{attribute 'object_name' := 'CycleStartDuty'}
METHOD PROTECTED CycleStartDuty : BOOL
// ----------------------------------------------------------------------------------
// cyclic actions outside of statemachine

// Simulation active
IF (SIf.stCfg.bolSimulation) THEN
	;
ELSE
	;
END_IF

// Cyclic call of the client connection
fbClientConnection();
// Cyclic call of method "HandleRxData"
THIS^.HandleRxData();

// Generate socket connected status info
IF (fbClientConnection.eState = eSOCKET_CONNECTED) THEN
	SIf.stStatus.bolSocketConnected:= TRUE;
ELSE
	SIf.stStatus.bolSocketConnected:= FALSE;	
	SIf.stStatus.bolComChecked:= FALSE;
END_IF

// Command close socket can be executed all the time.
// Used for error recovery in case if parent controller has an error.
IF (SIf.intCmd=cBCD_CMD_CLOSE_SOCKET) THEN	
	stStateMachine.intStateNext := cBCD_STA_CloseSocketBusy;
END_IF
			
SIf.strCmd := THIS^.getCmdState(intCmdState:=SIf.intCmd,bolState:=FALSE);
END_METHOD

{attribute 'object_name' := 'FB_init'}
METHOD FB_init : BOOL
VAR_INPUT
	///if TRUE, the retain variables are initialized (warm start / cold start)
	bInitRetains: BOOL;
	///if TRUE, the instance afterwards gets moved into the copy code (online change)
	bInCopyCode: BOOL;
END_VAR
// Communication Settings
SIf.stCfg.strSensorIPAdr := '192.168.1.103';  //'192.168.0.10'; 
SIf.stCfg.udiSensorPort := 9004;
SIf.stCfg.bolResponseIncludingDiagnostics := FALSE;
SIf.stCfg.iSensorType := E_BCD_Type.KEYENCE;

// Parameter
SIf.stPar.tTOConnection := T#50S;
SIf.stPar.tTOReceive := T#5S;
SIf.stPar.tTOSend := T#5S;
END_METHOD

{attribute 'object_name' := 'getCmdState'}
METHOD PROTECTED getCmdState : STRING
VAR_INPUT
	intCmdState: INT;
	bolState: BOOL;
END_VAR
// get string cmd/state string information in runtime
IF (bolState=FALSE) THEN
	
// cmd's
	CASE intCmdState OF
		cBCD_CMD_DONE: 
			getCmdState := 'cBCD_CMD_DONE';
		cBCD_CMD_CONNECT_SOCKET: 
			getCmdState := 'cBCD_CMD_CONNECT_SOCKET';
		cBCD_CMD_CLOSE_SOCKET: 
			getCmdState := 'cBCD_CMD_CLOSE_SOCKET';
		cBCD_CMD_READ_BARCODE: 
			getCmdState := 'cBCD_CMD_READ_BARCODE';		
		cBCD_CMD_COM_TEST: 
			getCmdState := 'cBCD_CMD_COM_TEST';			
	END_CASE;
ELSE

// state's
	CASE intCmdState OF
		cBCD_STA_WaitForJob: 
			getCmdState := 'cBCD_STA_WaitForJob';
		cBCD_STA_ConnectSocketBusy: 
			getCmdState := 'cBCD_STA_ConnectSocketBusy';
		cBCD_STA_CloseSocketBusy: 
			getCmdState := 'cBCD_STA_CloseSocketBusy';
		cBCD_STA_SocketClosed: 
			getCmdState := 'cBCD_STA_SocketClosed';	
		cBCD_STA_ReadCodeBusy: 
			getCmdState := 'cBCD_STA_ReadCodeBusy';	
		cBCD_STA_ComTestBusy:
			getCmdState := 'cBCD_STA_ComTestBusy';	
		cBCD_STA_Error: 
			getCmdState := 'cBCD_STA_Error';
	END_CASE;
	
END_IF
END_METHOD

{attribute 'object_name' := 'getSIf'}
METHOD getSIf : POINTER TO T_BCD
getSIf := ADR(SIf);
END_METHOD

{attribute 'object_name' := 'HandleRxData'}
METHOD PRIVATE HandleRxData
VAR
	uinI: UINT;
END_VAR
// GET/FETCH RX DATA
CASE intRxState OF
	
	// wait for read command
	cRxIdle:
		IF (bolExecuteRead=TRUE) AND (fbClientConnection.eState = eSOCKET_CONNECTED)THEN	

			// clear rx buffer
			FOR uinI:= 0 TO SIZEOF(aRxData)-1 DO
				aRxData[uinI]:= 16#00;
			END_FOR
			// Delete last message
			strReceivedMessage:= '';
			udiReceivedBytes := 0;
								
			// receive frame			
			fbReceive( bExecute := FALSE );
			fbReceive( 	sSrvNetId	:= '',
						hSocket		:= fbClientConnection.hSocket,
						cbLen		:= SIZEOF(aRxData),
						pDest		:= ADR(aRxData),
						bExecute	:= TRUE,
						tTimeout	:= SIf.stPar.tTOReceive);
			intRxState := cRxBusy;		
		END_IF
		
	// wait until receive not busy
	cRxBusy:
		fbReceive( bExecute := FALSE );
		IF NOT fbReceive.bBusy THEN
			IF NOT fbReceive.bError THEN
				IF (fbReceive.nRecBytes > 0) THEN (* some bytes received *)
					udiReceivedBytes := fbReceive.nRecBytes;
					intRxState := cRxConv; // convert received message
				ELSE
					// Try to read again
					intRxState := cRxIdle;
				END_IF	
			// Error	
			ELSE
				IF (SIf.stErr.bolErrorActive = FALSE) THEN
					SIf.stErr.bolErrorActive := TRUE;	
					SIf.stErr.udiErrorID := fbReceive.nErrId;	
					// Try to close the socket. Needs reconnect for socket after an error!	
					stStateMachine.intStateNext := cBCD_STA_CloseSocketBusy;	
				END_IF	
			END_IF			
		END_IF
			
	// convert received message to string
	cRxConv: 
		THIS^.PrepareReadMsg();
		THIS^.CheckSensorError(); // Error response: [STX]sFA <x>[ETX]    	
		bolExecuteRead:= FALSE; // Read done and data converted to string format
		intRxState := cRxIdle;
		
END_CASE
END_METHOD

{attribute 'object_name' := 'HandleTxData'}
METHOD PRIVATE HandleTxData
// HANDLE TX DATA
CASE intTxState OF
	
	// wait for send command (ready for send)
	cTxIdle:
		IF (bolExecuteSend) AND (fbClientConnection.eState = eSOCKET_CONNECTED)THEN									
			// send frame
			fbSend( bExecute := FALSE );
			fbSend(	sSrvNetID 	:= '',
					hSocket		:= fbClientConnection.hSocket,
					cbLen		:= rTxData.intMessageSize,
					pSrc		:= ADR(rTxData.aTxData),					// pointer to the frame data
					bExecute	:= TRUE,
					tTimeout 	:= SIf.stPar.tTOSend);
	
			intTxState := cTxBusy;							
		END_IF
		
	// wait until send not busy
	cTxBusy:
		fbSend( bExecute := FALSE );
		IF NOT (fbSend.bBusy) THEN
			intTxState := cTxIdle;
			// Check about FUB error	
			IF (fbSend.bError = TRUE) THEN
				IF (SIf.stErr.bolErrorActive = FALSE) THEN
					SIf.stErr.bolErrorActive := TRUE;	
					SIf.stErr.udiErrorID := fbSend.nErrId;	
					// Try to close the socket. Needs reconnect for socket after an error!	
					stStateMachine.intStateNext := cBCD_STA_CloseSocketBusy;	
				END_IF				
			// no error
			ELSE
				udiNSend := udiNSend + 1; // increment the number of send frames
				bolExecuteSend:= FALSE;
			END_IF
		END_IF
		
END_CASE
END_METHOD

{attribute 'object_name' := 'PrepareBarCodeData'}
METHOD PRIVATE PrepareBarCodeData
VAR
	intI: INT;
	intStartIndex: INT;
	intStartIndexCode: INT;
	bASCIISign: BYTE;
	strCharacter: STRING(1);
END_VAR

// Note: Currently only the bar code is read out from the received message. "OI=" section in message.
// Other data sections like e.g. "TT=", "OTL=", "CC=" are not prepared.

// ----------------------------------------------------
// Get bar code and write result to structure "stData"
// ----------------------------------------------------
	
// Example of message: <stx> <CR><LF> TT=125ms OTL=0mm CC=1 OI=25<CR><LF>45376049874<CR><LF> .... and so on ...   <etx>
				 
// Get start index for bar code 'OI='
intStartIndex := TC2_STANDARD.FIND(strReceivedMessage,'OI=');

// Loop over received message to get the bar code
FOR intI:=intStartIndex TO LEN(strReceivedMessage)-intStartIndex DO	
	// Convert to ASCII to detect CR and LF
	bASCIISign:= F_ToASC(Mid(strReceivedMessage,1,intI));
	// The bar code number starts after LF					
	IF (bASCIISign = cLF) THEN
		// Save start index of the bar code
		intStartIndexCode:= intI + 1;
	END_IF
	// Read every single number of the bar code until the end "CR"
	IF ((intStartIndexCode <> 0) AND (intI >= intStartIndexCode)) THEN
		// As long as the end is not reached...(The bar code number ends with CR)	
		IF (bASCIISign <> cCR) THEN								
			// Write result to structure stData	
			strCharacter:= Mid(strReceivedMessage,1,intI);
			SIf.stData.strBarCode:= CONCAT(SIf.stData.strBarCode,strCharacter);	
			SIf.stData.uliBarCode:= STRING_TO_ULINT(SIf.stData.strBarCode);
			SIf.stData.bolCodeReaded:= TRUE;																	
		ELSE
			// end of bar code reached "CR" -> EXIT loop
			EXIT;
		END_IF
	END_IF
	
END_FOR
END_METHOD

{attribute 'object_name' := 'PrepareReadMsg'}
METHOD PRIVATE PrepareReadMsg
VAR
	uinI: UINT;
	strCharacter: STRING(1);
END_VAR
// Delete last message
strReceivedMessage:= '';

// Loop over receive buffer
FOR uinI:= 0 TO SIZEOF(aRxData)-1 DO	
	// Start of text?
	IF (aRxData[uinI] = cSTX) THEN
		;
	// End of text?
	ELSIF (aRxData[uinI] = cETX) THEN
		EXIT;
	ELSE
		// Convert ASCII to string
		strCharacter:= F_ToCHR(aRxData[uinI]);
		strReceivedMessage:= CONCAT(strReceivedMessage,strCharacter);			
	END_IF
END_FOR
END_METHOD

{attribute 'object_name' := 'PrepareSendMsg'}
METHOD PRIVATE PrepareSendMsg
VAR_INPUT
	strMsg: STRING;
END_VAR
VAR
	intI: UINT;
	strCharacter: STRING(1);
END_VAR
// Clear send buffer
ClearTxBuffer();

// STX - start of telegramm
rTxData.aTxData[0]:= cSTX;

// Loop over message string and convert to ASCII
FOR intI:= 1 TO INT_TO_UINT(LEN(strMsg)) DO
	// Get char
	strCharacter:= MID(strMsg,1,UINT_TO_INT(intI));
	// Convert to ASCII
	rTxData.aTxData[intI]:= F_ToASC(strCharacter);
END_FOR

// ETX - end of telegramm
rTxData.aTxData[intI]:= cETX;

rTxData.intMessageSize := intI + 1;
END_METHOD

{attribute 'object_name' := 'sta_CloseSocketBusy'}
METHOD PROTECTED sta_CloseSocketBusy : BOOL
// state implemetation
//--------------------------------------------------------------------------------------
// Entry action
	IF (stStateMachine.intState<>stStateMachine.intStateLastCycle) THEN
		stStateMachine.intStateHistory := stStateMachine.intStateLastCycle;
		stStateMachine.intStateLastCycle := stStateMachine.intState;
		
		// Reset pending commands			
		bolExecuteSend:= FALSE;
		bolExecuteRead:= FALSE;
		// Reset Rx/Tx states
		intRxState:= cRxIdle;
		intTxState:= cTxIdle;
		// Close socket
		fbClientConnection.bEnable:= FALSE;

	END_IF

//--------------------------------------------------------------------------------------
// Cyclic action
	IF (stStateMachine.intState=stStateMachine.intStateLastCycle) THEN
		
	
		// State Change Condition

		// Check about FUB error	
		IF (fbClientConnection.bError = TRUE) OR (fbClientConnection.nErrId <> 0) THEN
			SIf.stErr.bolErrorActive := TRUE;	
			SIf.stErr.bolSocketError := TRUE;
			SIf.stErr.udiErrorID := fbClientConnection.nErrId;
			stStateMachine.intStateNext := cBCD_STA_Error;
		END_IF
	
		// Wait until socket is closed	
		IF (fbClientConnection.eState = eSOCKET_CLOSED) THEN
			stStateMachine.intStateNext := cBCD_STA_WaitForJob;
		ELSIF  (SIf.stErr.bolErrorActive= TRUE) THEN 
			stStateMachine.intStateNext := cBCD_STA_Error;		
		END_IF
	
	END_IF

//--------------------------------------------------------------------------------------
// Exit action
	IF (stStateMachine.intState<>stStateMachine.intStateNext) THEN
		SIf.intCmd := cBCD_CMD_DONE;
	END_IF
END_METHOD

{attribute 'object_name' := 'sta_ComTestBusy'}
METHOD PROTECTED sta_ComTestBusy : BOOL
// state implemetation
//--------------------------------------------------------------------------------------
// Entry action
	IF (stStateMachine.intState<>stStateMachine.intStateLastCycle) THEN
		stStateMachine.intStateHistory := stStateMachine.intStateLastCycle;
		stStateMachine.intStateLastCycle := stStateMachine.intState;

		// Clear data
		SIf.stData.stDevInfo.strComTestResult:='';
		SIf.stStatus.bolComChecked:=FALSE;
	
		// Init sub state machine
		stSubStateMachine.intState := cBCD_SUB_Send;
		stSubStateMachine.intStateNext := cBCD_SUB_Send;	
	END_IF

//--------------------------------------------------------------------------------------
// Cyclic action
	IF (stStateMachine.intState=stStateMachine.intStateLastCycle) THEN
			
		// sub state machine for reading the bar code	
		CASE stSubStateMachine.intState OF

			cBCD_SUB_Send:
				// Check Tx state idle
				IF (intTxState = cTxIdle) THEN
					CASE SIf.stCfg.iSensorType OF
						E_BCD_Type.SICK:
							THIS^.PrepareSendMsg('sRI0'); // Call SOPAS command "sRI0"
							
						E_BCD_Type.KEYENCE:
							THIS^.PrepareSendMsg('BCLR'); // clear send buffer
					END_CASE
					bolExecuteSend:= TRUE;
					stSubStateMachine.intState := cBCD_SUB_Wait;
				END_IF
		
			cBCD_SUB_Wait:
				// Wait until executed -> flag set back to false by method handle TxData
				IF (bolExecuteSend=FALSE)THEN
					stSubStateMachine.intState := cBCD_SUB_Read;
				END_IF
				
			cBCD_SUB_Read:
				// Check Rx state idle
				IF (intRxState = cRxIdle) THEN
					bolExecuteRead:= TRUE;
					stSubStateMachine.intState := cBCD_SUB_CheckAnswer;
				END_IF
			
			cBCD_SUB_CheckAnswer:
				// Wait until executed -> flag set back to false by method handle RxData
				IF (bolExecuteRead=FALSE)THEN				
					// Check about corresponding answer for the command	
					CASE SIf.stCfg.iSensorType OF
						E_BCD_Type.SICK:					
							IF (TC2_STANDARD.FIND(strReceivedMessage,'sRA') <> 0) THEN
								SIf.stData.stDevInfo.strComTestResult:=strReceivedMessage;
								SIf.stStatus.bolComChecked:=TRUE;
							END_IF
						
						E_BCD_Type.KEYENCE:
							IF (TC2_STANDARD.FIND(strReceivedMessage,'OK,BCLR') <> 0) THEN
								SIf.stData.stDevInfo.strComTestResult:=strReceivedMessage;
								SIf.stStatus.bolComChecked:=TRUE;
							END_IF
					END_CASE
					stSubStateMachine.intState := cBCD_SUB_Done;
				END_IF
			
			cBCD_SUB_Done:
				; // job executed
			
		END_CASE
		
		 // job executed
		IF (stSubStateMachine.intState = cBCD_SUB_Done) THEN
			stStateMachine.intStateNext := cBCD_STA_WaitForJob;	
		END_IF
	
	END_IF

//--------------------------------------------------------------------------------------
// Exit action
	IF (stStateMachine.intState<>stStateMachine.intStateNext) THEN
		SIf.intCmd := cBCD_CMD_DONE;
	END_IF
END_METHOD

{attribute 'object_name' := 'sta_ConnectSocketBusy'}
METHOD PROTECTED sta_ConnectSocketBusy : BOOL
// state implemetation
//--------------------------------------------------------------------------------------
// Entry action
	IF (stStateMachine.intState<>stStateMachine.intStateLastCycle) THEN
		stStateMachine.intStateHistory := stStateMachine.intStateLastCycle;
		stStateMachine.intStateLastCycle := stStateMachine.intState;
			
		// Initialize and connect socket
		fbClientConnection.nMode := CONNECT_MODE_ENABLEDBG; 			// not used
		fbClientConnection.sRemoteHost := SIf.stCfg.strSensorIPAdr;
		fbClientConnection.nRemotePort := SIf.stCfg.udiSensorPort;
		fbClientConnection.tReconnect := SIf.stPar.tTOConnection;
		fbClientConnection.bEnable:= TRUE;

	END_IF

//--------------------------------------------------------------------------------------
// Cyclic action
	IF (stStateMachine.intState=stStateMachine.intStateLastCycle) THEN
		
	
		// State Change Condition

		// Check about FUB error	
		IF (fbClientConnection.bError = TRUE) OR (fbClientConnection.nErrId <> 0) THEN
			SIf.stErr.bolErrorActive := TRUE;	
			SIf.stErr.bolSocketError := TRUE;
			SIf.stErr.udiErrorID := fbClientConnection.nErrId;
			stStateMachine.intStateNext := cBCD_STA_Error;
		END_IF
	
		// Wait for socket handle ID	
		IF (fbClientConnection.hSocket.handle <> 0) AND (fbClientConnection.eState = eSOCKET_CONNECTED) THEN
			stStateMachine.intStateNext := cBCD_STA_WaitForJob;
		END_IF

	END_IF

//--------------------------------------------------------------------------------------
// Exit action
	IF (stStateMachine.intState<>stStateMachine.intStateNext) THEN
		SIf.intCmd := cBCD_CMD_DONE;
	END_IF
END_METHOD

{attribute 'object_name' := 'sta_Error'}
METHOD PROTECTED sta_Error : BOOL
// state implemetation
//--------------------------------------------------------------------------------------
// Entry action
	IF (stStateMachine.intState<>stStateMachine.intStateLastCycle) THEN
		stStateMachine.intStateHistory := stStateMachine.intStateLastCycle;
		stStateMachine.intStateLastCycle := stStateMachine.intState;
		
		// Reset pending commands			
		bolExecuteSend:= FALSE;
		bolExecuteRead:= FALSE;
		// Reset Rx/Tx states
		intRxState:= cRxIdle;
		intTxState:= cTxIdle;
		
	END_IF


//--------------------------------------------------------------------------------------
// Cyclic action
	IF (stStateMachine.intState=stStateMachine.intStateLastCycle) THEN
			
		// State Change Condition
		IF (SIf.stErr.bolErrAck = TRUE) THEN
			// Reset all active errors
			SIf.stErr.bolErrorActive := FALSE;
			SIf.stErr.bolSocketError := FALSE;
			SIf.stErr.bolSensorError := FALSE;
			SIf.stErr.udiErrorID := 0;
			SIf.stErr.bolErrAck := FALSE;
			// Needs reconnect for socket after an error!		
			stStateMachine.intStateNext := cBCD_STA_CloseSocketBusy;		
		END_IF
		
	END_IF

//--------------------------------------------------------------------------------------
// Exit action
	IF (stStateMachine.intState<>stStateMachine.intStateNext) THEN
		;
	END_IF
END_METHOD

{attribute 'object_name' := 'sta_ReadCodeBusy'}
METHOD PROTECTED sta_ReadCodeBusy : BOOL
// state implemetation
//--------------------------------------------------------------------------------------
// Entry action
	IF (stStateMachine.intState<>stStateMachine.intStateLastCycle) THEN
		stStateMachine.intStateHistory := stStateMachine.intStateLastCycle;
		stStateMachine.intStateLastCycle := stStateMachine.intState;
		
		// Clear data
		SIf.stData.uliBarCode:=0;
		SIf.stData.strBarCode:='';
		SIf.stData.bolCodeReaded:= FALSE;
						
		// Init sub state machine
		stSubStateMachine.intState := cBCD_SUB_Send;
		stSubStateMachine.intStateNext := cBCD_SUB_Send;	
	END_IF

//--------------------------------------------------------------------------------------
// Cyclic action
	IF (stStateMachine.intState=stStateMachine.intStateLastCycle) THEN
			
		// sub state machine for reading the bar code	
		CASE stSubStateMachine.intState OF

			cBCD_SUB_Send:
				// Check Tx state idle
				IF (intTxState = cTxIdle) THEN
					CASE SIf.stCfg.iSensorType OF
						E_BCD_Type.SICK:
							THIS^.PrepareSendMsg('sMN mTCgateon'); // Call SOPAS method "sMN mTCgateon"
							bolExecuteSend:= TRUE;
							stSubStateMachine.intState := cBCD_SUB_Wait;
							
						E_BCD_Type.KEYENCE:
							THIS^.PrepareSendMsg('LON'); // Call Trigger ON
							bolExecuteSend:= TRUE;
							stSubStateMachine.intState := cBCD_SUB_Wait;
					ELSE
						SIf.stData.strBarCode:= 'no sensor type defined';
						SIf.stData.uliBarCode:= 0;
					END_CASE
					
				END_IF
		
			cBCD_SUB_Wait:
				// Wait until executed -> flag set back to false by method handle TxData
				IF (bolExecuteSend=FALSE)THEN
					stSubStateMachine.intState := cBCD_SUB_Read;
				END_IF
				
			cBCD_SUB_Read:
				// Check Rx state idle
				IF (intRxState = cRxIdle) THEN
					bolExecuteRead:= TRUE;
					stSubStateMachine.intState := cBCD_SUB_CheckAnswer;
				END_IF
			
			cBCD_SUB_CheckAnswer:
				// Wait until executed -> flag set back to false by method handle RxData
				IF (bolExecuteRead=FALSE)THEN				
					// Check about corresponding answer for the called method
					CASE SIf.stCfg.iSensorType OF
						E_BCD_Type.SICK:
							IF (FC_StrComp(strReceivedMessage,'sAN mTCgateon 1') = 0) THEN			
								// Check Rx state idle
								IF (intRxState = cRxIdle) THEN
									bolExecuteRead:= TRUE;
									stSubStateMachine.intState := cBCD_SUB_GetData;
								END_IF
							END_IF
							
						E_BCD_Type.KEYENCE:
							IF (FC_StrComp(strReceivedMessage,'OK,LON') = 0) THEN			
								// Check Rx state idle
								IF (intRxState = cRxIdle) THEN
									bolExecuteRead:= TRUE;
									stSubStateMachine.intState := cBCD_SUB_GetData;
								END_IF
							END_IF
					END_CASE
				END_IF
			
			cBCD_SUB_GetData:
				// Wait until executed -> flag set back to false by method handle RxData
				IF (bolExecuteRead=FALSE)THEN
					
					CASE SIf.stCfg.iSensorType OF
						E_BCD_Type.SICK:
							// No barcode recognized after the end of the time window ("duration" setting of sensor object trigger), NoRead !
							IF (((TC2_STANDARD.FIND(strReceivedMessage,'OI=') <> 0) OR NOT SIf.stCfg.bolResponseIncludingDiagnostics) 
								AND (TC2_STANDARD.FIND(strReceivedMessage,'*NoRead*') <> 0)) THEN			
								SIf.stData.strBarCode:='NoRead';
								stSubStateMachine.intState := cBCD_SUB_Done;
							END_IF
							
							// Barcode detected within the time window
							IF (((TC2_STANDARD.FIND(strReceivedMessage,'OI=') <> 0) OR NOT SIf.stCfg.bolResponseIncludingDiagnostics) 
								AND NOT (TC2_STANDARD.FIND(strReceivedMessage,'*NoRead*') <> 0)) THEN			
								// Prepare bar code data from received message
								THIS^.PrepareBarCodeData();
								stSubStateMachine.intState := cBCD_SUB_Done;
							END_IF
						
						E_BCD_Type.KEYENCE:
							// No barcode recognized after the end of the time window ("duration" setting of sensor object trigger), NoRead !
							IF (TC2_STANDARD.FIND(strReceivedMessage,'ERROR') <> 0) THEN			
								SIf.stData.strBarCode:='NoRead';
								stSubStateMachine.intState := cBCD_SUB_Done;
							END_IF
							
							// Barcode detected within the time window
							IF NOT (TC2_STANDARD.FIND(strReceivedMessage,'ERROR') <> 0) THEN			
								// Prepare bar code data from received message
								iStringLength := Tc2_Standard.LEN(strReceivedMessage);
								SIf.stData.strBarCode := Tc2_Standard.LEFT(strReceivedMessage,iStringLength-1);
								SIf.stData.uliBarCode:= STRING_TO_ULINT(SIf.stData.strBarCode);
								stSubStateMachine.intState := cBCD_SUB_Done;
							END_IF
					END_CASE
				END_IF
			
			cBCD_SUB_Done:
				; // job executed
			
		END_CASE
		
		 // job executed
		IF (stSubStateMachine.intState = cBCD_SUB_Done) THEN
			stStateMachine.intStateNext := cBCD_STA_WaitForJob;	
		END_IF
			
	END_IF

//--------------------------------------------------------------------------------------
// Exit action
	IF (stStateMachine.intState<>stStateMachine.intStateNext) THEN
		SIf.intCmd := cBCD_CMD_DONE;
	END_IF
END_METHOD

{attribute 'object_name' := 'sta_SocketClosed'}
METHOD PROTECTED sta_SocketClosed : BOOL
// state implemetation
//--------------------------------------------------------------------------------------
// Entry action
	IF (stStateMachine.intState<>stStateMachine.intStateLastCycle) THEN
		stStateMachine.intStateLastCycle := stStateMachine.intState;
		;
	END_IF

//--------------------------------------------------------------------------------------
// Cyclic action
	IF (stStateMachine.intState=stStateMachine.intStateLastCycle) THEN

		// State Change Condition
		IF (SIf.intCmd=cBCD_CMD_CONNECT_SOCKET) THEN
			stStateMachine.intStateNext := cBCD_STA_ConnectSocketBusy;
		END_IF
		
	END_IF

//--------------------------------------------------------------------------------------
// Exit action
	IF (stStateMachine.intState<>stStateMachine.intStateNext) THEN
		;
	END_IF
END_METHOD

{attribute 'object_name' := 'sta_WaitForJob'}
METHOD PROTECTED sta_WaitForJob : BOOL
// state implemetation
//--------------------------------------------------------------------------------------
// Entry action
	IF (stStateMachine.intState<>stStateMachine.intStateLastCycle) THEN
		stStateMachine.intStateLastCycle := stStateMachine.intState;
	END_IF


//--------------------------------------------------------------------------------------
// Cyclic action
	IF (stStateMachine.intState=stStateMachine.intStateLastCycle) THEN

		// State Change Condition
		IF (SIf.intCmd=cBCD_CMD_CONNECT_SOCKET) THEN						// Connect TCP socket
			stStateMachine.intStateNext := cBCD_STA_ConnectSocketBusy;
		ELSIF (SIf.intCmd=cBCD_CMD_CLOSE_SOCKET) THEN						// Close TCP socket
			stStateMachine.intStateNext := cBCD_STA_CloseSocketBusy;
		ELSIF (SIf.intCmd=cBCD_CMD_COM_TEST) THEN							// Communication test 
			stStateMachine.intStateNext := cBCD_STA_ComTestBusy;	
		ELSIF (SIf.intCmd=cBCD_CMD_READ_BARCODE) THEN						// Read bar code
			stStateMachine.intStateNext := cBCD_STA_ReadCodeBusy;				
		END_IF

				
	END_IF

//--------------------------------------------------------------------------------------
// Exit action
	IF (stStateMachine.intState<>stStateMachine.intStateNext) THEN
		;
	END_IF
END_METHOD

{attribute 'object_name' := 'StateMachine'}
METHOD PROTECTED StateMachine : BOOL

// main statemachine
CASE stStateMachine.intState OF	
	cBCD_STA_WaitForJob:
   		THIS^.sta_WaitForJob();
	cBCD_STA_ConnectSocketBusy: 
        THIS^.sta_ConnectSocketBusy();	
	cBCD_STA_CloseSocketBusy: 
        THIS^.sta_CloseSocketBusy();		
	cBCD_STA_SocketClosed: 
        THIS^.sta_SocketClosed();	
	cBCD_STA_ComTestBusy:
	    THIS^.sta_ComTestBusy();
	cBCD_STA_ReadCodeBusy:
	    THIS^.sta_ReadCodeBusy();
    cBCD_STA_Error: 
        THIS^.sta_Error();
END_CASE;
END_METHOD

END_FUNCTION_BLOCK

// POUs/Controller/Driver/BCD (Bar code driver)/FC_StrComp
FUNCTION FC_StrComp : DINT
VAR_INPUT
	strArg1: STRING(255);
	strArg2: STRING(255);
END_VAR
VAR
	stArg1: TC2_UTILITIES.T_Arg;
	stArg2: TC2_UTILITIES.T_Arg;
END_VAR


// String compare function use F_ARGCMP from beckhoff lib. TC2_UTILITIES

// set parameter for arg1
stArg1.cbLen:= INT_TO_UDINT(TC2_STANDARD.LEN(strArg1));
stArg1.pData:= ADR(strArg1);
stArg1.eType:= ARGTYPE_STRING;

// set parameter for arg2
stArg2.cbLen:= INT_TO_UDINT(TC2_STANDARD.LEN(strArg2));
stArg2.pData:= ADR(strArg2);
stArg2.eType:= ARGTYPE_STRING;

// call F_ARGCMP
FC_StrComp:= TC2_UTILITIES.F_ARGCMP(TRUE,stArg1,stArg2);

END_FUNCTION

// POUs/Controller/Driver/PRS [Present Sensor]/FB_PRS
FUNCTION_BLOCK FB_PRS EXTENDS FB_CtrlBase
VAR_INPUT
	In_bolPresent				: BOOL;
END_VAR
VAR_OUTPUT
	Out_bolPresent				: BOOL;
END_VAR
VAR
	/// Specific interface struct for public access
	SIf					: T_Ctrl_SIf_PRS;
END_VAR

(*__________________________________________________________________________________________________
¦	
¦	Vistaprint Schweiz GmbH
¦	CH - 8401 Winterthur
¦
¦	www.vistaprint.ch - info@vistaprint.ch
¦___________________________________________________________________________________________________

Function desription:
Vacuum Pump implementation. 


History:
Version		Date			Author		Comment
---------------------------------------------------------------------------------------------------
0.00.1		09.07.2013		PC			Start history
___________________________________________________________________________________________________*)


IF (me.bolActivate) THEN // cyclic call enabled
	IF (CIf.Info.bolInitDone=FALSE) THEN // first cycle -> init
		CtrlInit();
		CIf.Info.bolInitDone := TRUE;
	ELSE
		CycleStartDuty();
	
		Always();
		
		StateMachine();
		
		CycleEndDuty();
	END_IF
END_IF;

METHOD PROTECTED Always : BOOL
SUPER^.Always();

// ----------------------------------------------------------------------------------
// cyclic actions outside of statemachine
IF (me.StateMachine.intState<>cSTA_SINGLE_ANSWER) THEN
	
	; // always error supervision
	
END_IF

// ----------------------------------------------------------------------------------
// Conditions Always
IF (((me.Alarm.eActivAlmClass=E_AlmClass.EOFF) OR (me.Alarm.eActivAlmClass=E_AlmClass.OFF) OR (me.intCmd=cCMD_OFF))
		 AND (me.StateMachine.intState<>cSTA_ERROR) AND (me.StateMachine.intState<>cSTA_ERRORQuit) AND
		(me.StateMachine.intState<>cSTA_OFF) AND (me.StateMachine.intState<>cSTA_OFFBusy)) THEN
	// alarm evt EOFF, OFF or cmd off
	me.StateMachine.intStateNext := cSTA_OFFBusy;
END_IF
END_METHOD

PROPERTY PUBLIC CtrlSIf : POINTER TO T_CTRL_SIf_PRS
GET
CtrlSIf := ADR(SIf);
END_GET
END_PROPERTY

METHOD FB_init : BOOL
VAR_INPUT
	bInitRetains : BOOL; // if TRUE, the retain variables are initialized (warm start / cold start)
	bInCopyCode : BOOL;  // if TRUE, the instance afterwards gets moved into the copy code (online change)
END_VAR
VAR
	iIdx		: UINT;
	iLength		: UINT;	
END_VAR
//------------------------------------------------------------------------------------------------------------------------
// to manually change in new FUB implementation!!!
// define valid commands for this controller
iLength := SIZEOF(CIf.Job.aCmdList)/SIZEOF(CIf.Job.aCmdList[0]);
iIdx := 0;

WHILE (iIdx < iLength) AND (CIf.Job.aCmdList[iIdx].intCmd <> cCMD_INITIALIZED) DO
	iIdx := iIdx + 1; 
END_WHILE

IF (iIdx < iLength) THEN
// Add configuration of own comands	
	;
ELSE
	// Error if the aCmdList Array is to small
END_IF

// set name of class/typ
CIf.Info.strType := 'FB_PRS';
CIf.Info.strFullName := 'Present Sensor';

// set alarm class

//*******************************************************************************
// initial values
//*******************************************************************************

// software configuration
CIf.SwCfg.bolExist := TRUE;
CIf.SwCfg.bolEnable := TRUE;
CIf.SwCfg.bolSimulation :=  FALSE;

// parameter
SIf.Par.bolSimHangerAvailable := FALSE;
SIf.Par.udiDebounceAbsentTime_ms := 100;
SIf.Par.udiDebouncePresentTime_ms := 1500;
END_METHOD

METHOD PROTECTED getCmdState : STRING

VAR_INPUT
	intCmdState: INT;
	bolState: BOOL;
END_VAR
getCmdState := SUPER^.getCmdState(intCmdState:=intCmdState,bolState:=bolState); // get global/base defined cmds/states

IF (getCmdState='') THEN // global not defined get local
	// get string cmd/state string information in runtime
	IF (bolState=FALSE) THEN
		;
	ELSE
		// States's
		CASE intCmdState OF
			PRS_CmdState.cSTA_ABSENT: 
				getCmdState := 'cSTA_ABSENT';
			PRS_CmdState.cSTA_ABSENTBusy: 
				getCmdState := 'cSTA_ABSENTBusy';
			PRS_CmdState.cSTA_PRESENT: 
				getCmdState := 'cSTA_PRESENT';
			PRS_CmdState.cSTA_PRESENTBusy: 
				getCmdState := 'cSTA_PRESENTBusy';
		END_CASE;
	END_IF
END_IF
END_METHOD

METHOD getCtrlSIf : POINTER TO T_Ctrl_SIf_PRS
getCtrlSIf := ADR(SIf);
END_METHOD

METHOD PROTECTED IoInBridge : BOOL
// digitale and analoge inputs read from hardware or forcing
SIf.In.bolPresent.map := THIS^.In_bolPresent;

IF (CIf.SwCfg.bolSimulation = FALSE) THEN
	getInBol(CIf.Job.bolIoForce,ADR(SIf.In.bolPresent));
ELSE
	//simulation of global IO
END_IF
END_METHOD

METHOD PROTECTED IoOutBridge : BOOL
VAR
	bolSwitchValvesOff: BOOL;
END_VAR
// digitale and analoge inputs read from hardware or forcing
IF (CIf.SwCfg.bolSimulation = FALSE) THEN
//	setOutBol(CIf.Job.bolIoForce ,ADR(SIf.Out.bolClose));
	;
//	THIS^.Out_bolClose := SIf.Out.bolClose.map;
END_IF
END_METHOD

METHOD PROTECTED sta_ABSENT : BOOL
VAR_INPUT
END_VAR
// state implemetation
//--------------------------------------------------------------------------------------
// Entry action
	IF (me.StateMachine.intState<>me.StateMachine.intStateLastCycle) THEN
		me.StateMachine.intStateLastCycle := me.StateMachine.intState;
		THIS^.Out_bolPresent := FALSE;
	END_IF


//--------------------------------------------------------------------------------------
// Cyclic action
	IF (me.StateMachine.intState=me.StateMachine.intStateLastCycle) THEN
		IF CIf.SwCfg.bolSimulation THEN
			IF SIf.Par.bolSimHangerAvailable THEN
				me.StateMachine.intStateNext := PRS_CmdState.cSTA_PRESENTBusy;
			END_IF
		ELSE
			IF SIf.In.bolPresent.intern  THEN
				me.StateMachine.intStateNext := PRS_CmdState.cSTA_PRESENTBusy;
			END_IF;		
		END_IF
	END_IF


//--------------------------------------------------------------------------------------
// Exit action
	IF (me.StateMachine.intState<>me.StateMachine.intStateNext) THEN
		;
	END_IF
END_METHOD

METHOD PROTECTED sta_ABSENTBusy : BOOL
VAR_INPUT
END_VAR
// state implemetation
//--------------------------------------------------------------------------------------
// Entry action
	IF (me.StateMachine.intState<>me.StateMachine.intStateLastCycle) THEN
		me.StateMachine.intStateLastCycle := me.StateMachine.intState;
	END_IF


//--------------------------------------------------------------------------------------
// Cyclic action
	IF (me.StateMachine.intState=me.StateMachine.intStateLastCycle) THEN
		IF CIf.SwCfg.bolSimulation THEN
			IF SIf.Par.bolSimHangerAvailable THEN
				me.StateMachine.intStateNext := PRS_CmdState.cSTA_PRESENT;
			END_IF
		ELSE
			IF SIf.In.bolPresent.intern  THEN
				me.StateMachine.intStateNext := PRS_CmdState.cSTA_PRESENT;
			END_IF;		
			
			IF NOT SIf.In.bolPresent.intern AND (me.StateMachine.udiTimeInState_ms > SIf.Par.udiDebounceAbsentTime_ms) THEN
				me.StateMachine.intStateNext :=  PRS_CmdState.cSTA_ABSENT;
			END_IF
		END_IF
	END_IF


//--------------------------------------------------------------------------------------
// Exit action
	IF (me.StateMachine.intState<>me.StateMachine.intStateNext) THEN
		;
	END_IF
END_METHOD

METHOD PROTECTED sta_PON : BOOL
VAR_INPUT
END_VAR
// state implemetation
//--------------------------------------------------------------------------------------
// Entry action
	IF (me.StateMachine.intState<>me.StateMachine.intStateLastCycle) THEN
		me.StateMachine.intStateLastCycle := me.StateMachine.intState;
		
	END_IF


//--------------------------------------------------------------------------------------
// Cyclic action
	IF (me.StateMachine.intState=me.StateMachine.intStateLastCycle) THEN
		me.StateMachine.intStateNext := PRS_CmdState.cSTA_ABSENTBusy;
	END_IF




//--------------------------------------------------------------------------------------
// Exit action
	IF (me.StateMachine.intState<>me.StateMachine.intStateNext) THEN
		;
	END_IF
END_METHOD

METHOD PROTECTED sta_PRESENT : BOOL
VAR_INPUT
END_VAR
// state implemetation
//--------------------------------------------------------------------------------------
// Entry action
	IF (me.StateMachine.intState<>me.StateMachine.intStateLastCycle) THEN
		me.StateMachine.intStateLastCycle := me.StateMachine.intState;
		THIS^.Out_bolPresent := TRUE;
	END_IF


//--------------------------------------------------------------------------------------
// Cyclic action
	IF (me.StateMachine.intState=me.StateMachine.intStateLastCycle) THEN
		IF CIf.SwCfg.bolSimulation THEN
			IF NOT SIf.Par.bolSimHangerAvailable THEN
				me.StateMachine.intStateNext := PRS_CmdState.cSTA_ABSENTBusy;
			END_IF
		ELSE
			IF NOT SIf.In.bolPresent.intern  THEN
				me.StateMachine.intStateNext := PRS_CmdState.cSTA_ABSENTBusy;
			END_IF;		
		END_IF
	END_IF


//--------------------------------------------------------------------------------------
// Exit action
	IF (me.StateMachine.intState<>me.StateMachine.intStateNext) THEN
		;
	END_IF
END_METHOD

METHOD PROTECTED sta_PRESENTBusy : BOOL
VAR_INPUT
END_VAR
// state implemetation
//--------------------------------------------------------------------------------------
// Entry action
	IF (me.StateMachine.intState<>me.StateMachine.intStateLastCycle) THEN
		me.StateMachine.intStateLastCycle := me.StateMachine.intState;
	END_IF


//--------------------------------------------------------------------------------------
// Cyclic action
	IF (me.StateMachine.intState=me.StateMachine.intStateLastCycle) THEN
		IF CIf.SwCfg.bolSimulation THEN
			IF NOT SIf.Par.bolSimHangerAvailable THEN
				me.StateMachine.intStateNext := PRS_CmdState.cSTA_ABSENT;
			END_IF
		ELSE
			IF NOT SIf.In.bolPresent.intern  THEN
				me.StateMachine.intStateNext := PRS_CmdState.cSTA_ABSENT;
			END_IF;		
			
			IF SIf.In.bolPresent.intern AND (me.StateMachine.udiTimeInState_ms > SIf.Par.udiDebouncePresentTime_ms) THEN
				me.StateMachine.intStateNext :=  PRS_CmdState.cSTA_PRESENT;
			END_IF
		END_IF
	END_IF


//--------------------------------------------------------------------------------------
// Exit action
	IF (me.StateMachine.intState<>me.StateMachine.intStateNext) THEN
		;
	END_IF
END_METHOD

METHOD PROTECTED StateMachine : BOOL
SUPER^.StateMachine();

// main statemachine of base controller
CASE me.StateMachine.intState OF
    PRS_CmdState.cSTA_ABSENT: 
        THIS^.sta_ABSENT();
    PRS_CmdState.cSTA_ABSENTBusy: 
        THIS^.sta_ABSENTBusy();
    PRS_CmdState.cSTA_PRESENT: 
        THIS^.sta_PRESENT();
    PRS_CmdState.cSTA_PRESENTBusy: 
        THIS^.sta_PRESENTBusy();
END_CASE;
END_METHOD

END_FUNCTION_BLOCK

// POUs/Controller/Driver/RFD (RFID Driver)/FB_Com_3964R
FUNCTION_BLOCK FB_Com_3964R
VAR_INPUT
	/// Pointer to Received Data Array
	In_pRxData: POINTER TO ARRAY[0..255] OF BYTE;
	/// Pointer to Sending Data Array
	In_pTxData: POINTER TO ARRAY[0..255] OF BYTE;
	/// Amounth of sending data
	In_udiTxCount: UDINT;
	/// Error Acknowledge 
	In_bolErrorAck: BOOL;
END_VAR
VAR_IN_OUT
	/// Command to send Data 1=command; 0=Done
	InOut_bolSend: BOOL;
	/// Command Data received 1=received; 0=Done=Ready for next Data
	InOut_bolRec: BOOL;
END_VAR
VAR_OUTPUT
	/// Amounth of received data
	Out_udiRxCount: UDINT;
	/// Serial interface communication error
	Out_bolComError: BOOL;
	/// Error in protocoll procedure
	Out_bolProtocolErr: BOOL;
	/// Error information to master
	Out_udiErrorCode: UDINT;
END_VAR
VAR
	In_stEL6inData AT %I*: TC2_SERIALCOM.EL6inData22B;
	Out_stEL6outData AT %Q*: TC2_SERIALCOM.EL6outData22B;
	/// Internal Variables
	udiI: UDINT;
	/// Local variable for loops
	udiK: UDINT;
	/// Internal Error Reset
	bolIntReset: BOOL;
	/// Count call trials
	uinCountCall: UINT;
	/// Count call Retrys
	uinCountRetry: UINT;
	/// Temporary value for cecking the sum
	bytCheckValue: BYTE;
	/// Antenna is initializied, until it is not initializied, it send 16#02 in all possible baudrates
	bolSLGInitialized: BOOL := FALSE;
	/// Check Timeout
	bolTimeout: BOOL;
	/// Check Timeout
	bolWait: BOOL;
	/// Send NAK needed
	bolSendNAK: BOOL;
	/// Receive Wait signs
	timWaitReceive: TIME := TIME#5ms;
	/// Receive Wait signs
	timWaitAck: TIME := TIME#400ms;
	/// Sign delay time
	timZVZ: TIME := TIME#45ms;
	/// Time ACK delay
	timQVZ: TIME := TIME#145ms;
	/// Initialisation of the HW card
	bolInitRequest: BOOL;
	/// Setting of the HW Card
	bolSendContinious: BOOL;
	/// Priority at RFID
	bolPriority: BOOL;
	/// Send DLE doubletimes
	bolDLEDouble: BOOL;
	/// New data received
	bolComDataReceived: BOOL;
	/// receiving busy
	bolComRecBusy: BOOL;
	/// Received Data
	udiComSizeReceiveData: UDINT;
	/// Sending busy
	bolComSendBusy: BOOL;
	/// Error at serial line control
	bolErrSerialLineControl: BOOL;
	/// Error at serial line control
	stErrSerialLineControl: ComError_t;
	/// Error at serial line  receiving data
	bolErrReceive: BOOL;
	/// Error at serial line  receiving data
	stErrReceive: ComError_t;
	/// Error at serial line sending data
	bolErrSend: BOOL;
	/// Error at serial line sending data
	stErrSend: ComError_t;
	/// Define Buffer for preparations
	aRxData: ARRAY[0..255] OF BYTE;
	aTxData: ARRAY[0..255] OF BYTE;
	/// Define Buffer for Funciton
	stRxBuffer: TC2_SERIALCOM.ComBuffer;
	/// Transmit data buffer; used with all receive function blocks 
	stTxBuffer: TC2_SERIALCOM.ComBuffer;
	/// Sub Statemachine
	intState: INT := 0;
	intStateOld: INT := 0;
	udiStateLoop: UDINT;
	a_intStateHist: ARRAY[0..9] OF INT;
	udiStateDebug: UDINT;
	udiStateDebugMax: UDINT;
	/// Function for serial communication
	fbSerialLineControl: TC2_SERIALCOM.SerialLineControl;
	fbSerialReceiveData: TC2_SERIALCOM.ReceiveData;
	fbSerialSendData: TC2_SERIALCOM.SendData;
	fbSerialClearComBuffer: TC2_SERIALCOM.ClearComBuffer;
	fbTon: TC2_STANDARD.TON;
	fbWait: TC2_STANDARD.TON;
	fbZVZ: TC2_STANDARD.TON;
	fbQVZ: TC2_STANDARD.TON;
	fbPriority: TC2_STANDARD.TON;
END_VAR
VAR CONSTANT
	cSTX: USINT := 16#2;
	cDLE: USINT := 16#10;
	cETX: USINT := 16#3;
	cNAK: USINT := 16#15;
	/// Startup
	cRFD_3964_Start: INT := 2500;
	/// Startup
	cRFD_3964_Init: INT := 2501;
	/// Wait for Job
	cRFD_3964_Wait: INT := 2502;
	/// Read recived sign
	cRFD_3964_RxRead: INT := 2504;
	/// Ackn. receiving ready
	cRFD_3964_RxReadRdy: INT := 2506;
	/// Recive Data
	cRFD_3964_RxData: INT := 2508;
	/// Achn. received Data
	cRFD_3964_RxCheckData: INT := 2510;
	/// Send Ack to Slave
	cRFD_3964_RxAck: INT := 2512;
	/// Send Ack to Slave
	cRFD_3964_RxAck2: INT := 2514;
	/// Send Request to Slave
	cRFD_3964_TxRequest: INT := 2550;
	/// Send Wait answer
	cRFD_3964_TxWait: INT := 2552;
	/// Send Data
	cRFD_3964_TxSend: INT := 2554;
	/// Send Wait for Ack
	cRFD_3964_TxAck: INT := 2556;
	/// Error
	cRFD_3964_Error: INT := 2580;
END_VAR

(*__________________________________________________________________________________________________
¦	
¦	Vistaprint Schweiz GmbH
¦	CH - 8401 Winterthur
¦
¦	www.vistaprint.ch - info@vistaprint.ch
¦___________________________________________________________________________________________________

Function desription:
Driver for communication protocoll 3964R
Description in Siemens manual from CP341, A5E02191070-03


History:
Version		Date			Author		Comment
---------------------------------------------------------------------------------------------------
0.00.1		23.07.2013		AVME/PRE	Start history
___________________________________________________________________________________________________*)

// Always
fbSerialLineControl(
	Mode:= TC2_SERIALCOM.ComSerialLineMode_t.SERIALLINEMODE_EL6_22B, 
	pComIn:= ADR(In_stEL6inData), 
	pComOut:= ADR(Out_stEL6outData), 
	SizeComIn:= SIZEOF(In_stEL6inData), 
	Error=> bolErrSerialLineControl, 
	ErrorID=> stErrSerialLineControl, 
	TxBuffer:= stTxBuffer, 
	RxBuffer:= stRxBuffer);
	
// Check timers
IF intState >= cRFD_3964_Wait THEN
	fbZVZ(PT:= timZVZ);
	fbQVZ(PT:= timQVZ);
	fbWait(PT:= timWaitAck);

	// Check priority
	fbPriority(IN:= bolPriority, PT:=timWaitAck);
	IF (fbPriority.Q = TRUE) THEN
		bolPriority := FALSE;
	END_IF

END_IF
		
// Startup set correct Step
IF intState < cRFD_3964_Start THEN
	intState := cRFD_3964_Start;
END_IF

// State Machine
CASE intState OF
	cRFD_3964_Start:
		// Clear Buffer
		FOR udiI := 0 TO SIZEOF(aRxData)-1 DO
			aRxData[udiI] := 0;
			aTxData[udiI] := 0;
		END_FOR
		bolSLGInitialized := FALSE;
		
		// Clear counters
		uinCountCall := 0;
		uinCountRetry := 0;
		
		bolInitRequest := FALSE;
		bolSendContinious := FALSE;
		
		
		// Next State
		IF (bolErrSerialLineControl = FALSE) AND (bolTimeout=TRUE) THEN
			intState := cRFD_3964_Init;
		ELSIF (bolErrSerialLineControl = TRUE) THEN
			intState := cRFD_3964_Error;
		END_IF

	// Wait for a job or received Data //	
	cRFD_3964_Init:	
		bolInitRequest := TRUE;
		
		IF (bolErrSerialLineControl = FALSE) AND ((In_stEL6inData.Status.2 = TRUE) OR (bolTimeout=TRUE)) THEN	// Initialisation Done  OR (bolTimeout=TRUE)
			intState := cRFD_3964_Wait;
		ELSIF (bolErrSerialLineControl = TRUE) THEN
			intState := cRFD_3964_Error;
		END_IF
	
	// Wait for a job or received Data //	
	cRFD_3964_Wait:	
		bolInitRequest := FALSE;
		bolSendNAK := FALSE;
		fbZVZ.IN := FALSE;
		fbQVZ.IN := FALSE;
		fbWait.IN := FALSE;
		
		fbSerialReceiveData(
		//	pPrefix:= , // Not used because no prefix in telegram
			LenPrefix:= 0, 
		//	pSuffix:= , // Not used because no suffix in telegram
			LenSuffix:= 0, 
			pReceiveData:= ADR(aRxData), 
			SizeReceiveData:= 255, 
			Timeout:= timWaitReceive, 
		//	Reset:= , 
			DataReceived=> bolComDataReceived, 
			busy=> bolComRecBusy, 
			Error=> stErrReceive, 
			RxTimeout=> bolErrReceive, 
			LenReceiveData=> udiComSizeReceiveData, 
			RXbuffer:= stRxBuffer);
		
		//Check if Data is received
		IF bolComDataReceived = TRUE THEN
			intState := cRFD_3964_RxRead;
		ELSIF (InOut_bolSend = TRUE) AND (bolPriority = FALSE) THEN
			intState := cRFD_3964_TxRequest;
		END_IF
			
	// Read first signs if new data sending needed //	
	cRFD_3964_RxRead: 
		// Check reached Sign
		// Send ready for reach Data if STX is send and Buffer is ready to use
		fbWait.IN := TRUE;
		IF (((aRxData[0] = cSTX) OR (bolSLGInitialized = FALSE))  AND (InOut_bolRec = FALSE)) THEN 
			aTxData[0] := cDLE;
		ELSE
			aTxData[0] := cNAK;
		END_IF
		
		IF ((fbWait.Q = FALSE) OR (InOut_bolRec = TRUE)) THEN
			intState := cRFD_3964_RxReadRdy; 
			fbWait.IN := FALSE; 
		END_IF
		
	// Send Feedback //		
	cRFD_3964_RxReadRdy:
		fbZVZ.IN := TRUE; 

		IF fbZVZ.Q = TRUE THEN
			fbSerialSendData(
				pSendData:= ADR(aTxData), 
				Length:= 1, 
				Busy=> bolComSendBusy, 
				Error=> stErrSend, 
				TXbuffer:= stTxBuffer);
				bolSendContinious := TRUE;
		END_IF
			
		// Check transition
		IF (bolComSendBusy = FALSE) AND (bolSLGInitialized = TRUE) AND (fbZVZ.Q = TRUE) THEN		// AND (stErrSend = 0)
			IF (aTxData[0] = cDLE) THEN
				intState := cRFD_3964_RxData;
			ELSE
				intState := cRFD_3964_Wait;
			END_IF
		ELSIF ((bolComSendBusy = TRUE) OR (bolTimeout = TRUE)) AND (uinCountCall < 10) AND (fbZVZ.Q = TRUE) THEN
			uinCountCall := uinCountCall + 1;
			intState := cRFD_3964_Wait;
		ELSIF ((bolComSendBusy = TRUE) OR (bolTimeout = TRUE)) AND (fbZVZ.Q = TRUE) THEN
			bolSendNAK := TRUE;
			intState := cRFD_3964_Error;
		END_IF
		
	// Read Data //	
	cRFD_3964_RxData:
		fbZVZ.IN := FALSE; 
		fbSerialReceiveData(
		//	pPrefix:= , // Not used because no prefix in telegram
			LenPrefix:= 0, 
		//	pSuffix:= , // Not used because no suffix in telegram
			LenSuffix:= 0, 
			pReceiveData:= ADR(aRxData), 
			SizeReceiveData:= 255, 
			Timeout:= timWaitReceive, 
		//	Reset:= , 
			DataReceived=> bolComDataReceived, 
			busy=> bolComRecBusy, 
			Error=> stErrReceive, 
			RxTimeout=> bolErrReceive, 
			LenReceiveData=> udiComSizeReceiveData, 
			RXbuffer:= stRxBuffer);
				
		IF (bolComDataReceived = TRUE) AND (bolComRecBusy = FALSE) AND (udiComSizeReceiveData <= 255)  THEN
			intState := cRFD_3964_RxCheckData;
		ELSIF ((bolTimeout = TRUE) OR (udiComSizeReceiveData > 255)) THEN	 // OR (stErrReceive <> 0)
			bolSendNAK := TRUE;
			IF (uinCountCall < 10) THEN
				uinCountCall := uinCountCall + 1;
				intState := cRFD_3964_RxAck;
			ELSE
				intState := cRFD_3964_Error;
			END_IF
		END_IF
	
	// Check Received Data //	
	cRFD_3964_RxCheckData:
		//minimal 1 Byte, ETX and BCC   	ETX is last sign for BCC					DLE is last sign for ETX
		IF (udiComSizeReceiveData >= 4) THEN
			IF ((aRxData[udiComSizeReceiveData-2] = cETX) AND (aRxData[udiComSizeReceiveData-3] = cDLE)) THEN
				// Check BCC
				bytCheckValue := aRxData[0] XOR aRxData[1];
				FOR udiI := 2 TO  (udiComSizeReceiveData-2) DO
					bytCheckValue := bytCheckValue XOR aRxData[udiI];
				END_FOR
				
				IF (bytCheckValue = aRxData[udiComSizeReceiveData-1]) THEN //BCC OK
					// Copy Data
					FOR udiI := 0 TO (SIZEOF(aRxData)-1) DO
						In_pRxData^[udiI] := 0;
					END_FOR
					udiK := 0;
					FOR udiI := 0 TO udiComSizeReceiveData-4 DO
						In_pRxData^[udiK] := aRxData[udiI];
						IF (aRxData[udiI] = cDLE) AND (aRxData[udiI+1] = cDLE) THEN		// DLE Doubling, only take on DLE
							udiI := udiI+1;
						END_IF
						udiK := udiK + 1;
					END_FOR
					InOut_bolRec := TRUE;
					intState := cRFD_3964_RxAck;
				ELSE
					bolSendNAK := TRUE;				
					IF (uinCountCall < 10) THEN
						uinCountCall := uinCountCall + 1;
						intState := cRFD_3964_RxAck;
					ELSE
						intState := cRFD_3964_Error;
					END_IF
				END_IF
			ELSE
				bolSendNAK := TRUE;				
				IF (uinCountCall < 10) THEN
					uinCountCall := uinCountCall + 1;
					intState := cRFD_3964_RxAck;
				ELSE
					intState := cRFD_3964_Error;
				END_IF
			END_IF
		ELSIF aRxData[0] = cSTX THEN
			aTxData[0] := cDLE;
			intState := cRFD_3964_RxReadRdy;
		ELSE
			bolSendNAK := TRUE;				
			IF (uinCountCall < 10) THEN
				uinCountCall := uinCountCall + 1;
				intState := cRFD_3964_RxAck;
			ELSE
				intState := cRFD_3964_Error;
			END_IF
		END_IF
	// SEND Acknowledge of received Data //
	cRFD_3964_RxAck:
		IF bolSendNAK = TRUE THEN
			aTxData[0] := cNAK;
		ELSE
			aTxData[0] := cDLE;
		END_IF
		
		fbZVZ.IN := TRUE; // Prepare for send step
		fbSerialSendData(
			pSendData:= ADR(aTxData), 
			Length:= 1, 
			Busy=> bolComSendBusy, 
			Error=> stErrSend, 
			TXbuffer:= stTxBuffer);
				
					
		// Check transition
		IF (bolComSendBusy = FALSE) AND (stErrSend = 0) AND (bolSendNAK = FALSE) THEN	//  AND (fbZVZ.Q = TRUE)
			uinCountCall := 0;
			bolSLGInitialized := TRUE;
			intState := cRFD_3964_Wait;
		ELSIF (bolComSendBusy = FALSE) AND (stErrSend = 0) AND (bolSendNAK = TRUE) THEN	//  AND (fbZVZ.Q = TRUE)
			intState := cRFD_3964_Wait;
		END_IF

	// SEND Acknowledge of received Data //
	cRFD_3964_RxAck2:
		IF bolSendNAK = TRUE THEN
			aTxData[0] := cNAK;
		ELSE
			aTxData[0] := cDLE;
		END_IF
		
		fbSerialSendData(
			pSendData:= ADR(aTxData), 
			Length:= 1, 
			Busy=> bolComSendBusy, 
			Error=> stErrSend, 
			TXbuffer:= stTxBuffer);
				
		// Check transition
		IF (bolComSendBusy = FALSE) AND (stErrSend = 0) AND (bolSendNAK = FALSE) AND (bolWait = TRUE) THEN
			uinCountCall := 0;
			bolSLGInitialized := TRUE;
			intState := cRFD_3964_Wait;
		ELSIF (bolComSendBusy = FALSE) AND (stErrSend = 0) AND (bolSendNAK = TRUE) AND (bolWait = TRUE) THEN
			intState := cRFD_3964_Wait;
		ELSIF ((bolComSendBusy = TRUE) OR (bolTimeout = TRUE)) THEN
			intState := cRFD_3964_Error;
		END_IF

/////////////////////////////////////////////////////////////////////
// Sending Data
	// Request a sending job at Slave //
	cRFD_3964_TxRequest:
		aTxData[0] := cSTX;
		fbSerialSendData(
			pSendData:= ADR(aTxData), 
			Length:= 1, 
			Busy=> bolComSendBusy, 
			Error=> stErrSend, 
			TXbuffer:= stTxBuffer);
		bolSendContinious := TRUE;
			
		// Check transition
		IF (bolComSendBusy = FALSE) AND (stErrSend = 0) THEN
			intState := cRFD_3964_TxWait;
		ELSIF ((bolComSendBusy = TRUE) OR (bolTimeout = TRUE)) THEN
			intState := cRFD_3964_Error;
		END_IF
		
	// Wait for answer ready //	
	cRFD_3964_TxWait:	
		fbSerialReceiveData(
		//	pPrefix:= , // Not used because no prefix in telegram
			LenPrefix:= 0, 
		//	pSuffix:= , // Not used because no suffix in telegram
			LenSuffix:= 0, 
			pReceiveData:= ADR(aRxData), 
			SizeReceiveData:= 1, 
			Timeout:= timWaitReceive, 
		//	Reset:= , 
			DataReceived=> bolComDataReceived, 
			busy=> bolComRecBusy, 
			Error=> stErrReceive, 
			RxTimeout=> bolErrReceive, 
			LenReceiveData=> udiComSizeReceiveData, 
			RXbuffer:= stRxBuffer);
				
		IF (bolComDataReceived = TRUE) AND (bolComRecBusy = FALSE) AND (udiComSizeReceiveData <= 255)  THEN
			IF aRxData[0] = cDLE THEN
				intState := cRFD_3964_TxSend;
			ELSIF aRxData[0] = cSTX THEN	// At Start of Text 
				intState := cRFD_3964_RxRead;
				bolPriority := TRUE;
			ELSE
				IF uinCountRetry > 10 THEN
					intState := cRFD_3964_Error;
				ELSE 
					uinCountRetry := uinCountRetry + 1;
					intState := cRFD_3964_Wait;
				END_IF
			END_IF			
		ELSIF ((bolTimeout = TRUE) OR (udiComSizeReceiveData > 255)) THEN
			IF uinCountCall > 10 THEN
				intState := cRFD_3964_Error;
			ELSE
				IF bolSLGInitialized = TRUE THEN
					uinCountCall := uinCountCall + 1;
					intState := cRFD_3964_Wait;
				END_IF
			END_IF				
		END_IF
	
	// sending data //	
	cRFD_3964_TxSend:
		//only prepare data if not sending //
		IF (bolComSendBusy = FALSE) THEN
			bolDLEDouble := FALSE;
			udiI := 11;
			FOR udiI := 0 TO (SIZEOF(aTxData)-1) DO
				aTxData[udiI] := 0;
			END_FOR
			udiI := 0;
			udiK := 0;
			FOR udiK := 0 TO In_udiTxCount-1 DO
				aTxData[udiI] := In_pTxData^[udiK];
				IF aTxData[udiI] = cDLE THEN
					udiI := udiI + 1;
					aTxData[udiI] := cDLE;
					bolDLEDouble := TRUE;
				END_IF
				udiI := udiI + 1;				
			END_FOR
			aTxData[udiI] := cDLE;
			udiI := udiI + 1;
			//IF bolDLEDouble = TRUE THEN		// DLE Doubling at the end of the data if once uced as data
			//	aTxData[udiI] := cDLE;
			//	udiI := udiI + 1;				
			//END_IF
			aTxData[udiI] := cETX;
			
			bytCheckValue := aTxData[0] XOR aTxData[1];
			FOR udiK := 2 TO  udiI DO
				bytCheckValue := bytCheckValue XOR aTxData[udiK];
			END_FOR
			udiI := udiI + 1;
			aTxData[udiI] := bytCheckValue;
			udiI := udiI + 1;
		END_IF

		fbSerialSendData(
			pSendData:= ADR(aTxData), 
			Length:= udiI, 
			Busy=> bolComSendBusy, 
			Error=> stErrSend, 
			TXbuffer:= stTxBuffer);
			
		// Check transition
		IF (bolComSendBusy = FALSE) AND (stErrSend = 0) THEN
			intState := cRFD_3964_TxAck;
		ELSIF ((bolComSendBusy = TRUE) OR (bolTimeout = TRUE)) THEN
			IF uinCountRetry > 10 THEN
				intState := cRFD_3964_Error;
			ELSE 
				uinCountRetry := uinCountRetry + 1;
				intState := cRFD_3964_Wait;
			END_IF
		END_IF
		
	// Wait for answer ready //	
	cRFD_3964_TxAck:
		fbSerialReceiveData(
		//	pPrefix:= , // Not used because no prefix in telegram
			LenPrefix:= 0, 
		//	pSuffix:= , // Not used because no suffix in telegram
			LenSuffix:= 0, 
			pReceiveData:= ADR(aRxData), 
			SizeReceiveData:= 255, 
			Timeout:= timWaitReceive, 
		//	Reset:= , 
			DataReceived=> bolComDataReceived, 
			busy=> bolComRecBusy, 
			Error=> stErrReceive, 
			RxTimeout=> bolErrReceive, 
			LenReceiveData=> udiComSizeReceiveData, 
			RXbuffer:= stRxBuffer);
				
		IF (bolComDataReceived = TRUE) AND (bolComRecBusy = FALSE) AND (udiComSizeReceiveData <= 255)  THEN
			IF aRxData[0] = cDLE THEN
				intState := cRFD_3964_Wait;
				InOut_bolSend := FALSE;
				bolSLGInitialized := TRUE;
			ELSE
				IF uinCountRetry > 10 THEN
					intState := cRFD_3964_Error;
				ELSE 
					uinCountRetry := uinCountRetry + 1;
					intState := cRFD_3964_Wait;
				END_IF
			END_IF			
		ELSIF ((bolTimeout = TRUE) OR (udiComSizeReceiveData > 255)) THEN	 // OR (stErrReceive <> 0)
			IF uinCountRetry > 10 THEN
				intState := cRFD_3964_Error;
			ELSE
				uinCountRetry := uinCountRetry + 1;
				intState := cRFD_3964_Wait;
			END_IF				
		END_IF
	

////////////////////////////////////////////////////////////		
		// Error State //
		cRFD_3964_Error:
			// Send correct information
			IF bolErrSerialLineControl = TRUE THEN
				Out_udiErrorCode := INT_TO_UDINT(stErrSerialLineControl);
				Out_bolComError := TRUE;
			ELSIF bolErrSend = TRUE THEN
				Out_udiErrorCode := INT_TO_UDINT(stErrSend);				
				Out_bolComError := TRUE;
			ELSIF bolTimeout = TRUE THEN
				Out_bolProtocolErr := TRUE;
			ELSIF (Out_bolComError = FALSE) AND (Out_bolProtocolErr = FALSE) THEN
				Out_bolComError := TRUE;
			END_IF
			
			// Send NAK to RFID Reader
			IF bolSendNAK = TRUE THEN
				aTxData[0] := cNAK;
				fbSerialSendData(
					pSendData:= ADR(aTxData), 
					Length:= 1, 
					Busy=> bolComSendBusy, 
					Error=> stErrSend, 
					TXbuffer:= stTxBuffer);
					
				IF bolComSendBusy = FALSE THEN
					bolSendNAK := FALSE;
				END_IF
			END_IF
			
			// Acknowledge reset Error bit and informations
			IF (In_bolErrorAck = TRUE) OR (bolIntReset=TRUE) THEN
				intState := cRFD_3964_Wait;
				bolSendNAK := FALSE;
				bolErrSerialLineControl := FALSE; 
				bolErrReceive := FALSE;
				bolErrSend := FALSE;
				bolTimeout := FALSE;
				Out_udiErrorCode := 0;
				Out_bolComError := FALSE;
				Out_bolProtocolErr := FALSE;
				uinCountCall := 0;
				uinCountRetry := 0;
				bolIntReset := FALSE;
				In_bolErrorAck := FALSE;
				bolInitRequest := FALSE;
				InOut_bolRec := FALSE;
				InOut_bolSend := FALSE;
				bolSLGInitialized := FALSE;
			END_IF
		
END_CASE

// Write parallel Outputs to commando word
//Out_stEL6outData.Ctrl.2 := bolInitRequest;
Out_stEL6outData.Ctrl.3 := bolSendContinious;

// make History of States
IF intStateOld <> intState THEN
	udiStateLoop := 9;
	WHILE udiStateLoop > 0 DO
		a_intStateHist[udiStateLoop] := a_intStateHist[udiStateLoop-1];
		udiStateLoop := udiStateLoop-1;
	END_WHILE
	a_intStateHist[0] := intState;
	intStateOld := intState;
	// Time Out control
	// Check timeout
	fbTon(IN:= FALSE, PT:= timQVZ, Q=>bolTimeout );
ELSE
	IF intState <> cRFD_3964_Error THEN
		fbTon(IN:= TRUE, PT:= timQVZ, Q=>bolTimeout );
	END_IF
END_IF

END_FUNCTION_BLOCK

// POUs/Controller/Driver/RFD (RFID Driver)/FB_ExCom
FUNCTION_BLOCK FB_ExCom
VAR_INPUT
	/// Pointer to Received Data Array
	In_pRxData: POINTER TO ARRAY[0..255] OF BYTE;
	/// Pointer to Sending Data Array
	In_pTxData: POINTER TO ARRAY[0..255] OF BYTE;
	/// Amounth of sending data
	In_udiTxCount: UDINT;
	/// Error Acknowledge 
	In_bolErrorAck: BOOL;
END_VAR
VAR_IN_OUT
	/// Command to send Data 1=command; 0=Done
	InOut_bolSend: BOOL;
	/// Command Data received 1=received; 0=Done=Ready for next Data
	InOut_bolRec: BOOL;
END_VAR
VAR_OUTPUT
	/// Amounth of received data
	Out_udiRxCount: UDINT;
	/// Serial interface communication error
	Out_bolComError: BOOL;
	/// Error in protocoll procedure
	Out_bolProtocolErr: BOOL;
	/// Error information to master
	Out_udiErrorCode: UDINT;
END_VAR
VAR
	In_stEL6inData AT %I*: TC2_SERIALCOM.EL6inData22B;
	Out_stEL6outData AT %Q*: TC2_SERIALCOM.EL6outData22B;
	/// Internal Variables
	udiI: UDINT;
	/// Local variable for loops
	udiK: UDINT;
	/// Internal Error Reset
	bolIntReset: BOOL;
	/// Count call trials
	uinCountCall: UINT;
	/// Count call Retrys
	uinCountRetry: UINT;
	/// Temporary value for cecking the sum
	bytCheckValue: BYTE;
	/// Antenna is initializied, until it is not initializied, it send 16#02 in all possible baudrates
	bolSLGInitialized: BOOL := FALSE;
	/// Check Timeout
	bolTimeout: BOOL;
	/// Check Timeout
	bolWait: BOOL;
	/// Send NAK needed
	bolSendNAK: BOOL;
	/// Receive Wait signs
	timWaitReceive: TIME := TIME#5ms;
	/// Receive Wait signs
	timWaitAck: TIME := TIME#400ms;
	/// Sign delay time
	timZVZ: TIME := TIME#45ms;
	/// Time ACK delay
	timQVZ: TIME := TIME#145ms;
	/// Initialisation of the HW card
	bolInitRequest: BOOL;
	/// Setting of the HW Card
	bolSendContinious: BOOL;
	/// Priority at RFID
	bolPriority: BOOL;
	/// Send DLE doubletimes
	bolDLEDouble: BOOL;
	/// New data received
	bolComDataReceived: BOOL;
	/// receiving busy
	bolComRecBusy: BOOL;
	/// Received Data
	udiComSizeReceiveData: UDINT;
	/// Sending busy
	bolComSendBusy: BOOL;
	/// Error at serial line control
	bolErrSerialLineControl: BOOL;
	/// Error at serial line control
	stErrSerialLineControl: ComError_t;
	/// Error at serial line  receiving data
	bolErrReceive: BOOL;
	/// Error at serial line  receiving data
	stErrReceive: ComError_t;
	/// Error at serial line sending data
	bolErrSend: BOOL;
	/// Error at serial line sending data
	stErrSend: ComError_t;
	/// Define Buffer for preparations
	aRxData: ARRAY[0..255] OF BYTE;
	aTxData: ARRAY[0..255] OF BYTE;
	/// Define Buffer for Funciton
	stRxBuffer: TC2_SERIALCOM.ComBuffer;
	/// Transmit data buffer; used with all receive function blocks 
	stTxBuffer: TC2_SERIALCOM.ComBuffer;
	/// Sub Statemachine
	intState: INT := 0;
	intStateOld: INT := 0;
	udiStateLoop: UDINT;
	a_intStateHist: ARRAY[0..9] OF INT;
	udiStateDebug: UDINT;
	udiStateDebugMax: UDINT;
	/// Function for serial communication
	fbSerialLineControl: TC2_SERIALCOM.SerialLineControl;
	fbSerialReceiveData: TC2_SERIALCOM.ReceiveData;
	fbSerialSendData: TC2_SERIALCOM.SendData;
	fbTon: TC2_STANDARD.TON;
	fbWait: TC2_STANDARD.TON;
END_VAR
VAR CONSTANT
	/// Startup
	cExCom_Start: INT := 2500;
	/// Startup
	cExCom_Init: INT := 2501;
	/// Wait for Job
	cExCom_Wait: INT := 2502;
	/// Read recived sign
	cExCom_RxRead: INT := 2504;
	/// Send Data
	cExCom_TxPrepare: INT := 2550;
	/// Send Data
	cExCom_TxSend: INT := 2552;
	/// Error
	cExCom_Error: INT := 2580;
END_VAR

(*__________________________________________________________________________________________________
¦	
¦	Vistaprint Schweiz GmbH
¦	CH - 8401 Winterthur
¦
¦	www.vistaprint.ch - info@vistaprint.ch
¦___________________________________________________________________________________________________

Function desription:
Driver for communication protocoll 3964R
Description in Siemens manual from CP341, A5E02191070-03


History:
Version		Date			Author		Comment
---------------------------------------------------------------------------------------------------
0.00.1		23.07.2013		AVME/PRE	Start history
___________________________________________________________________________________________________*)

// Always
fbSerialLineControl(
	Mode:= TC2_SERIALCOM.ComSerialLineMode_t.SERIALLINEMODE_EL6_22B, 
	pComIn:= ADR(In_stEL6inData), 
	pComOut:= ADR(Out_stEL6outData), 
	SizeComIn:= SIZEOF(In_stEL6inData), 
	Error=> bolErrSerialLineControl, 
	ErrorID=> stErrSerialLineControl, 
	TxBuffer:= stTxBuffer, 
	RxBuffer:= stRxBuffer);
	
// Check timers
IF intState >= cExCom_Wait THEN
	fbWait(PT:= timWaitAck);
END_IF
		
// Startup set correct Step
IF intState < cExCom_Start THEN
	intState := cExCom_Start;
END_IF

// State Machine
CASE intState OF
	cExCom_Start:
		// Clear Buffer
		FOR udiI := 0 TO 255 DO
			aRxData[udiI] := 0;
			aTxData[udiI] := 0;
		END_FOR
		bolSLGInitialized := FALSE;
		
		// Clear counters
		uinCountCall := 0;
		uinCountRetry := 0;
		
		bolInitRequest := FALSE;
		bolSendContinious := FALSE;
		
		
		// Next State
		IF (bolErrSerialLineControl = FALSE) AND (bolTimeout=TRUE) THEN
			intState := cExCom_Init;
		ELSIF (bolErrSerialLineControl = TRUE) THEN
			intState := cExCom_Error;
		END_IF

	// Wait for a job or received Data //	
	cExCom_Init:	
		bolInitRequest := TRUE;
		
		IF (bolErrSerialLineControl = FALSE) AND (bolTimeout=TRUE) THEN	// Initialisation Done
			intState := cExCom_Wait;
		ELSIF (bolErrSerialLineControl = TRUE) THEN
			intState := cExCom_Error;
		END_IF
	
	// Wait for a job or received Data //	
	cExCom_Wait:	
		bolInitRequest := FALSE;
		bolSendNAK := FALSE;
		fbWait.IN := FALSE;
		
		fbSerialReceiveData(
		//	pPrefix:= , // Not used because no prefix in telegram
			LenPrefix:= 0, 
		//	pSuffix:= , // Not used because no suffix in telegram
			LenSuffix:= 0, 
			pReceiveData:= ADR(aRxData), 
			SizeReceiveData:= 255, 
			Timeout:= timWaitReceive, 
		//	Reset:= , 
			DataReceived=> bolComDataReceived, 
			busy=> bolComRecBusy, 
			Error=> stErrReceive, 
			RxTimeout=> bolErrReceive, 
			LenReceiveData=> udiComSizeReceiveData, 
			RXbuffer:= stRxBuffer);
		
		//Check if Data is received
		IF bolComDataReceived = TRUE THEN
			intState := cExCom_RxRead;
		ELSIF (InOut_bolSend = TRUE) AND (bolPriority = FALSE) THEN
			intState := cExCom_TxPrepare;
		END_IF
			
	// Read first signs if new data sending needed //	
	cExCom_RxRead: 
		// Read Signs
		IF (udiComSizeReceiveData >0) THEN
			// Copy Data
			FOR udiI := 0 TO (SIZEOF(aRxData)-1) DO
				In_pRxData^[udiI] := 0;
			END_FOR
			FOR udiI := 0 TO udiComSizeReceiveData-1 DO
				In_pRxData^[udiI] := aRxData[udiI];
			END_FOR
			InOut_bolRec := TRUE;
			Out_udiRxCount := udiComSizeReceiveData;
		END_IF
		
		intState := cExCom_Wait;

		
	// Send Data //		
	cExCom_TxPrepare:
		FOR udiI := 0 TO (SIZEOF(aTxData)-1) DO
			aTxData[udiI] := 0;
		END_FOR
		FOR udiI := 0 TO In_udiTxCount-1 DO
			aTxData[udiI] := In_pTxData^[udiI];
		END_FOR
		intState := cExCom_TxSend;

	cExCom_TxSend:	
		fbSerialSendData(
			pSendData:= ADR(aTxData), 
			Length:= In_udiTxCount, 
			Busy=> bolComSendBusy, 
			Error=> stErrSend, 
			TXbuffer:= stTxBuffer);
			bolSendContinious := TRUE;

			
		// Check transition
		IF (bolComSendBusy = FALSE) AND (stErrSend = 0) THEN
			intState := cExCom_Wait;
			InOut_bolSend := FALSE;
		ELSIF ((bolComSendBusy = TRUE) AND (bolTimeout = TRUE)) OR (stErrSend <> 0) THEN
			bolErrSend := TRUE;
			intState := cExCom_Error;
		END_IF
		

////////////////////////////////////////////////////////////		
		// Error State //
		cExCom_Error:
			IF bolErrSerialLineControl = TRUE THEN
				Out_udiErrorCode := INT_TO_UDINT(stErrSerialLineControl);
				Out_bolComError := TRUE;
			ELSIF bolErrSend = TRUE THEN
				Out_udiErrorCode := INT_TO_UDINT(stErrSend);				
				Out_bolComError := TRUE;
			ELSIF bolTimeout = TRUE THEN
				Out_bolProtocolErr := TRUE;
			ELSIF (Out_bolComError = FALSE) AND (Out_bolProtocolErr = FALSE) THEN
				Out_bolComError := TRUE;
			END_IF
		
			
			IF (In_bolErrorAck = TRUE) OR (bolIntReset=TRUE) THEN
				intState := cExCom_Wait;
				bolErrSerialLineControl := FALSE; 
				bolErrReceive := FALSE;
				bolErrSend := FALSE;
				bolTimeout := FALSE;
				Out_udiErrorCode := 0;
				Out_bolComError := FALSE;
				Out_bolProtocolErr := FALSE;
				uinCountCall := 0;
				uinCountRetry := 0;
				In_bolErrorAck := FALSE;
				bolInitRequest := FALSE;
			END_IF
		
END_CASE

// Write parallel Outputs to commando word
//Out_stEL6outData.Ctrl.2 := bolInitRequest;
//Out_stEL6outData.Ctrl.3 := bolSendContinious;

// make History of States
IF intStateOld <> intState THEN
	udiStateLoop := 9;
	WHILE udiStateLoop > 0 DO
		a_intStateHist[udiStateLoop] := a_intStateHist[udiStateLoop-1];
		udiStateLoop := udiStateLoop-1;
	END_WHILE
	a_intStateHist[0] := intState;
	intStateOld := intState;
	// Time Out control
	// Check timeout
	fbTon(IN:= FALSE, PT:= timQVZ, Q=>bolTimeout );
ELSE
	IF intState <> cExCom_Error THEN
		fbTon(IN:= TRUE, PT:= timQVZ, Q=>bolTimeout );
	END_IF
END_IF

END_FUNCTION_BLOCK

// POUs/Controller/Driver/RFD (RFID Driver)/FB_HEXSTRING_TO_ULINT
FUNCTION FB_HEXSTRING_TO_ULINT : ULINT
VAR_INPUT
	in_strSTRING: STRING;
END_VAR
VAR
	uinLenght: UINT;
	intI: INT;
	uliFact: ULINT;
	usiSign: USINT;
	uliReturn: ULINT;
	ausiTemp: ARRAY[0..15] OF USINT;
END_VAR

uinLenght := INT_TO_UINT(TC2_STANDARD.LEN(in_strSTRING));
uliReturn := 0;

IF (uinLenght > 16) THEN
	FB_HEXSTRING_TO_ULINT := 0;
	
ELSE
	MEMCPY(destAddr:=ADR(ausiTemp), srcAddr:=ADR(in_strSTRING), n:=uinLenght);		// COPY to buffer
	intI := UINT_TO_INT(uinLenght)-1;
	uliFact := 1;
	WHILE intI >= 0 DO
		IF (ausiTemp[intI] >= 16#30) AND (ausiTemp[intI] <= 16#39) THEN		// 0=16#30 ...9=16#39
			usiSign := ausiTemp[intI] - 16#30;
		ELSIF (ausiTemp[intI] >= 16#41) AND (ausiTemp[intI] <= 16#46) THEN		// A=16#41 ...F=16#46
			usiSign := ausiTemp[intI] - 55;
		ELSIF (ausiTemp[intI] >= 16#61) AND (ausiTemp[intI] <= 16#66) THEN		// a=16#61 ...f=16#66
			usiSign := ausiTemp[intI] - 87;
		ELSE
			FB_HEXSTRING_TO_ULINT := 0;
			RETURN;
		END_IF
		
		uliReturn := uliReturn + usiSign * uliFact;
		intI := intI - 1;
		uliFact := uliFact * 16;
	END_WHILE
		
END_IF

	FB_HEXSTRING_TO_ULINT := uliReturn;

END_FUNCTION

// POUs/Controller/Driver/RFD (RFID Driver)/FB_RFD
FUNCTION_BLOCK FB_RFD
VAR
	bolActivate: BOOL := TRUE;
	bolInitDone: BOOL;
	bolInitComDone: BOOL;
	bolFB_ComError: BOOL;	// communication FB has a error
	///Communication sending is busy to the serial Card
	bolComSend: BOOL;
	/// Size of Sendingdata
	udiComSizeSendData: UDINT;
	///Communication Data Received
	bolComDataReceived: BOOL;
	/// Size of received Data from serial interface
	udiComSizeReceiveData: UDINT;
	///Sdo Setting is busy to the serial Card
	bolSdoBusy: BOOL;
	///Sdo Setting executing
	bolSdoExecute: BOOL;
	/// Antenna Job done
	bolAntennaJobDone: BOOL;
	/// Job Reading is done
	bolReadDone: BOOL;
	/// Job Writing is done
	bolWriteDone: BOOL;
	/// Job Reset SLG is done
	bolResetJobDone: BOOL;
	/// Job Reset SLG has Error
	bolResetJobError: BOOL;
	/// Job Read SLG State is done
	bolSLGJobDone: BOOL;
	/// Job Read SLG State is done
	bolMDSJobDone: BOOL;
	/// Information to SDO Error
	udiSdoErrorNbr: UDINT;
	/// Information to Communication over 3964 protocol Error
	udi3964R_Error_Nbr: UDINT;
	/// Count Reset cycles
	udiResetCount: UDINT;
	/// Count Job Tryals
	udiJobCount: UDINT;
	/// Time in State ms
	udiTimeInState_ms: UDINT;
	/// State information from RF ID Tag
	bytRFIDState: BYTE;
	/// driver specific interface
	SIf: T_RFD;
	/// get direct Buffer from Interface
	/// access over mapping!! {attribute 'TcLinkTo':='TIID^Device 1 (EtherCAT)^Box 1 (SGDV-E1 CoE Drive)^2nd Transmit PDO mapping^Status word'}
	aRxData: ARRAY[0..255] OF BYTE;
	aTxData: ARRAY[0..255] OF BYTE;
	/// Function for serial communication
	fbEcCoeSdoWrite: TC2_ETHERCAT.FB_EcCoESdoWrite;
	fbCom_3964R: FB_Com_3964R;
	stStateMachine: T_RFD_StateMachine;
	stSubStateMachine: T_RFD_StateMachine;
	///case variable
	usiCase: USINT;
	///case variable for service cmd's
	usiCaseScmd: USINT;
	/// help values for parameter handling
	sinValue: SINT;
	intValue: INT;
	dinValue: DINT;
	usiValue: USINT;
	uinValue: UINT;
	udiValue: UDINT;
	udiI: UDINT;
	udiLoopBuffer: UDINT;
	udiLoopData: UDINT;
	udiLoopSend: UDINT;
	fbTimeoutState: TON;

END_VAR

(*__________________________________________________________________________________________________
¦	
¦	Vistaprint Schweiz GmbH
¦	CH - 8401 Winterthur
¦
¦	www.vistaprint.ch - info@vistaprint.ch
¦___________________________________________________________________________________________________

Function desription:
Driver for Simatic RFID Reader and Writer RF310R 6GT2801-1AB10


History:
Version		Date			Author		Comment
---------------------------------------------------------------------------------------------------
0.00.1		09.07.2013		AVME/PRE	Start history
0.00.2		24.09.2013		AVME/KVO	Parameter init from element controller to driver
___________________________________________________________________________________________________*)


IF (bolActivate) THEN // cyclic call enabled
	
	IF (bolInitDone=FALSE) THEN // first cycle -> init
		CtrlInit();
		bolInitDone := TRUE;
	ELSE
		CycleStartDuty();
		
		StateMachine_Service(); // handles asynchron service commands
		
		StateMachine();
		
		CycleEndDuty();
	END_IF
	
END_IF;

METHOD PROTECTED CtrlInit : BOOL
// one time first cyclic call
;
END_METHOD

METHOD PROTECTED CycleEndDuty : BOOL
SIf.strState := THIS^.getCmdState(intCmdState:=stStateMachine.intState,bolState:=TRUE);

IF (stStateMachine.intState<>stStateMachine.intStateNext) THEN
	stStateMachine.intState := stStateMachine.intStateNext;  // set next state for next cycle
END_IF

(***************************************************************
        Function Block Calls
***************************************************************)
END_METHOD

METHOD PROTECTED CycleStartDuty : BOOL
// ----------------------------------------------------------------------------------
// cyclic actions outside of statemachine
fbCom_3964R(
	In_pRxData:= ADR(aRxData), 
	In_pTxData:= ADR(aTxData), 
	In_udiTxCount:= udiComSizeSendData, 
	In_bolErrorAck:= SIf.stErr.bolErrAck, 
	InOut_bolSend:= bolComSend, 
	InOut_bolRec:= bolComDataReceived, 
	Out_udiRxCount=> udiComSizeReceiveData, 
	Out_bolComError=> bolFB_ComError, 
	Out_bolProtocolErr=> SIf.stErr.bolProtcolError, 
	Out_udiErrorCode=> udi3964R_Error_Nbr);

	IF bolFB_ComError = TRUE THEN
		SIf.stErr.bolComError := TRUE;
		SIf.stErr.udiErrorID := udi3964R_Error_Nbr;
	END_IF
(* program code at the beginning of each PLC cycle *)
IF bolInitComDone=TRUE THEN
	// Received Data checking and interpreting
	IF bolComDataReceived = TRUE THEN
		CASE aRxData[1] OF
			0:		//16#00 Startup Telegram OR Reset
				IF aRxData[0]= 16#02 THEN 	// Startup Telegram
					IF aRxData[1]= 16#0F THEN
						SIf.stStatus.bolStartupOk := TRUE;				
					END_IF
				ELSE		// Reset Acknowledge
					SIf.stStatus.stSLG_State.worFWVersion := aRxData[3];
					bytRFIDState := aRxData[2];	// Stetebyte copy 1:1
					IF aRxData[2]= 16#00 THEN
						bolResetJobDone := TRUE;
					ELSE
						bolResetJobError := TRUE;
					END_IF
				END_IF
			15:		//16#0F RFID Tag present state
				bytRFIDState := aRxData[2];	// Stetebyte copy 1:1
				IF bytRFIDState=0 THEN
					IF aRxData[4]>0 THEN
						SIf.stStatus.bolPresent := TRUE;
					ELSE
						SIf.stStatus.bolPresent := FALSE;
					END_IF
				END_IF
			1, 65:		//16#01 16#61 Write Acknowledge
				bytRFIDState := aRxData[2];	// Stetebyte copy 1:1
				IF bytRFIDState=0 THEN
					bolWriteDone := TRUE;
				ELSE
					SIf.stErr.bolRFIDError := TRUE;
				END_IF
			2, 66:		//16#02 16#42 Read Acknowledge
				bytRFIDState := aRxData[2];	// Stetebyte copy 1:1
				IF (bytRFIDState=0) AND (SIf.stCur.uinAdressData+SIf.stCur.usiCount <= 255) AND (SIf.stCur.usiCount+6 <= 255) THEN		// AND (SIf.stCur.usiCount = (aRxData[0]-5))
					FOR udiLoopBuffer := 0 TO (SIf.stCur.usiCount) DO
						SIf.stCur.pData^[SIf.stCur.uinAdressData+udiLoopBuffer] := aRxData[udiLoopBuffer+6];
					END_FOR	
					bolReadDone := TRUE;
				ELSE
					SIf.stErr.bolRFIDError := TRUE;
				END_IF
			4, 68:		//16#04 16#44 SLG State
				bytRFIDState := aRxData[2];	// Statebyte copy 1:1
				IF bytRFIDState<>0 THEN
					SIf.stErr.bolRFIDError := TRUE;
				ELSE
					IF aRxData[3]=16#01 THEN		// SLG State mode 1
						// HW Type
						SIf.stStatus.stSLG_State.bytHWType := aRxData[4];
						// HW Version
						SIf.stStatus.stSLG_State.worHWVersion := 0;
						SIf.stStatus.stSLG_State.worHWVersion := aRxData[5];
						SIf.stStatus.stSLG_State.worHWVersion := SHL(SIf.stStatus.stSLG_State.worHWVersion,8);
						SIf.stStatus.stSLG_State.worHWVersion := SIf.stStatus.stSLG_State.worHWVersion OR aRxData[6];
						// URL Version
						SIf.stStatus.stSLG_State.worURLVersion := 0;
						SIf.stStatus.stSLG_State.worURLVersion := aRxData[7];
						SIf.stStatus.stSLG_State.worURLVersion := SHL(SIf.stStatus.stSLG_State.worURLVersion,8);
						SIf.stStatus.stSLG_State.worURLVersion := SIf.stStatus.stSLG_State.worURLVersion OR aRxData[8];
						// FW Type
						SIf.stStatus.stSLG_State.bytFWType := aRxData[9];
						// FW Version
						SIf.stStatus.stSLG_State.worFWVersion := 0;
						SIf.stStatus.stSLG_State.worFWVersion := aRxData[10];
						SIf.stStatus.stSLG_State.worFWVersion := SHL(SIf.stStatus.stSLG_State.worFWVersion,8);
						SIf.stStatus.stSLG_State.worFWVersion := SIf.stStatus.stSLG_State.worFWVersion OR aRxData[11];
						// TR Type
						SIf.stStatus.stSLG_State.bytDriverType := aRxData[12];
						// TR Version
						SIf.stStatus.stSLG_State.worDriverVersion := 0;
						SIf.stStatus.stSLG_State.worDriverVersion := aRxData[13];
						SIf.stStatus.stSLG_State.worDriverVersion := SHL(SIf.stStatus.stSLG_State.worDriverVersion,8);
						SIf.stStatus.stSLG_State.worDriverVersion := SIf.stStatus.stSLG_State.worDriverVersion OR aRxData[14];
						// Serial Interface
						SIf.stStatus.stSLG_State.bytComm := aRxData[15];
						// Serial Interface Baud Rate
						SIf.stStatus.stSLG_State.bytBaud := aRxData[16];
						// sending power (only RF380R)
						SIf.stStatus.stSLG_State.bytPower := aRxData[20];
						// Number of maximal tags in the field
						SIf.stStatus.stSLG_State.bytMtag := aRxData[21];
						// air interface 0=RF300; 1=ISO generall; 3=ISO infineon Chip; 4=ISO Fujitsu; 5=ISO NXP; 6=ISO TI; 7=ISO ST
						SIf.stStatus.stSLG_State.bytFtim := aRxData[23];
						// State antenna 1=ON; 2=OFF
						SIf.stStatus.stSLG_State.bytAntenna := aRxData[25];
						// Tag presence 0=No presence; 1=prexence
						SIf.stStatus.stSLG_State.bytPresence := aRxData[27];
					ELSE		// SLG Diagnose Mode 6
						// Errorcounter inactive mode
						SIf.stStatus.stSLG_Diag.usiFZP := aRxData[4];
						// Counter abort
						SIf.stStatus.stSLG_Diag.usiABZ := aRxData[5];
						// Errorcounter code errors
						SIf.stStatus.stSLG_Diag.usiCFZ := aRxData[6];
						// Errorcounter signature errors
						SIf.stStatus.stSLG_Diag.usiSFZ := aRxData[7];
						// Errorcounter CRC
						SIf.stStatus.stSLG_Diag.usiCRCFZ := aRxData[8];
						// Actual command state
						SIf.stStatus.stSLG_Diag.usiBSTAT := aRxData[9];
						// Counter interface errors to host (Parity, BCC, Frame)
						SIf.stStatus.stSLG_Diag.usiASMFZ := aRxData[10];
					END_IF
				END_IF
				bolSLGJobDone := TRUE;

			11, 75:		//16#0B 16#4B MDS State
				bytRFIDState := aRxData[2];	// Statebyte copy 1:1
				IF bytRFIDState<>0 THEN
					SIf.stErr.bolRFIDError := TRUE;
				ELSE
					// UID
					SIf.stStatus.abyteUID[7] := aRxData[4];
					SIf.stStatus.abyteUID[6] := aRxData[5];
					SIf.stStatus.abyteUID[5] := aRxData[6];
					SIf.stStatus.abyteUID[4] := aRxData[7];
					SIf.stStatus.abyteUID[3] := aRxData[8];
					SIf.stStatus.abyteUID[2] := aRxData[9];
					SIf.stStatus.abyteUID[1] := aRxData[10];
					SIf.stStatus.abyteUID[0] := aRxData[11];
						
					IF aRxData[3]=16#01 THEN		// MDS State mode 1 RF300
						SIf.stStatus.stMDS_State.bytMDSType := aRxData[12];
						SIf.stStatus.stMDS_State.bytLockState := aRxData[13];
						SIf.stStatus.stMDS_State.worMemSize := 0;		// No information at this type			
						SIf.stStatus.stMDS_State.bytLockState := 0;		// No information at this type
						SIf.stStatus.stMDS_State.bytBlockSize := 0;		// No information at this type
						SIf.stStatus.stMDS_State.bytBlockNo := 0;		// No information at this type
					ELSIF aRxData[3]=16#02 THEN		// MDS Diagnose mode 2 RF300
						SIf.stStatus.stMDS_Diag.usiLFD := aRxData[12];
						SIf.stStatus.stMDS_Diag.usiFZP := aRxData[13];
						SIf.stStatus.stMDS_Diag.usiFZA := aRxData[14];
						SIf.stStatus.stMDS_Diag.usiANWZ := aRxData[15];
					ELSIF aRxData[3]=16#03 THEN		// MDS State mode 3 ISO
						SIf.stStatus.stMDS_State.bytMDSType := aRxData[12];
						SIf.stStatus.stMDS_State.bytVersion := aRxData[13];
						SIf.stStatus.stMDS_State.worMemSize := aRxData[14]*256 + aRxData[15];				
						SIf.stStatus.stMDS_State.bytLockState := aRxData[16];
						SIf.stStatus.stMDS_State.bytBlockSize := aRxData[17];
						SIf.stStatus.stMDS_State.bytBlockNo := aRxData[18];
					END_IF
				END_IF
				bolMDSJobDone := TRUE;
		
					
			10, 42:		//16#2A SET Antenna
				bytRFIDState := aRxData[2];	// Stetebyte copy 1:1
				IF bytRFIDState=0 THEN
					bolAntennaJobDone := TRUE;
				ELSE
					SIf.stErr.bolRFIDError := TRUE;
					SIf.stErr.udiErrorID := 1000 + bytRFIDState;
			END_IF
			16#FF:		//Communication Check to SLG
				SIf.stStatus.bolL_UEB := TRUE;		
		
		END_CASE
	// Data processed, reset bol to ACK
	bolComDataReceived := FALSE;
	END_IF
END_IF

// always go to Error 
(*KVO no auto start because config write from RFW-slow programm
IF (stStateMachine.intState<cRFD_STA_PowerOnBusy) AND (stStateMachine.intState<>cRFD_STA_Error) THEN
	stStateMachine.intStateNext := cRFD_STA_PowerOnBusy;
ELS*)
IF SIf.stCfg.bolSimulation = TRUE THEN
	SIf.intCmd := cSTA_DONE;
ELSIF (SIf.stErr.bolErrorActive) AND 
	(stStateMachine.intState<>cRFD_STA_Error)  THEN
	stStateMachine.intStateNext := cRFD_STA_Error;
// always go to PowerOff 
ELSIF ((SIf.intCmd=cRFD_CMD_CTRL_OFF)) AND 
	(stStateMachine.intState<>cRFD_STA_Off) AND 
	(stStateMachine.intState<>cRFD_STA_Error) THEN
	stStateMachine.intStateNext := cRFD_STA_Off;
ELSIF ((SIf.intCmd=RFD_Cmd.cRFD_CMD_CTRL_ON) AND (stStateMachine.intState<>cRFD_STA_PowerOnBusy)) THEN
	stStateMachine.intStateNext := cRFD_STA_PowerOnBusy;
END_IF

SIf.strCmd := THIS^.getCmdState(intCmdState:=SIf.intCmd,bolState:=FALSE);
END_METHOD

METHOD FB_init : BOOL
VAR_INPUT
	///if TRUE, the retain variables are initialized (warm start / cold start)
	bInitRetains: BOOL;
	///if TRUE, the instance afterwards gets moved into the copy code (online change)
	bInCopyCode: BOOL;
END_VAR
VAR
	udiTaskCnt: UDINT;
	ii: UINT;
END_VAR
SIf.intCmd := cRFD_CMD_DONE;
SIf.intServiceCmd := cRFD_CMD_DONE; // not used at the moment
stStateMachine.intStateLastCycle  := cRFD_CMD_DONE; //EntryStop of power BASE_PLC.OFF enable

// Vaild Values into the Configuration
SIf.stCfg.usiFtimSetting := E_Typ_Ftim.RF300;

// Communication Settings
SIf.stCfg.eTyp := E_Typ_RFW.RF310R;
SIf.stCfg.uinBaudrate := INT_TO_USINT(E_Typ_Baudrate.baud_57600);
SIf.stCfg.stNetId := '192.168.70.26.3.1';
SIf.stCfg.uinSlaveAddr := 1002;
END_METHOD

METHOD PROTECTED getCmdState : STRING
VAR_INPUT
	intCmdState: INT;
	bolState: BOOL;
END_VAR
// get string cmd/state string information in runtime
IF (bolState=FALSE) THEN
	// cmd's
	CASE intCmdState OF
		cRFD_CMD_DONE: 
			getCmdState := 'cRFD_CMD_DONE';
		cRFD_CMD_CTRL_ON: 
			getCmdState := 'cRFD_CMD_CTRL_ON';
		cRFD_CMD_CTRL_OFF: 
			getCmdState := 'cRFD_CMD_CTRL_OFF';
		cRFD_CMD_Write: 
			getCmdState := 'cRFD_CMD_Write';
		cRFD_CMD_Read: 
			getCmdState := 'cRFD_CMD_Read';
		cRFD_CMD_MDS: 
			getCmdState := 'cRFD_CMD_MDS';
		cRFD_CMD_SLG: 
			getCmdState := 'cRFD_CMD_SLG';
	END_CASE;
ELSE

// States
	CASE intCmdState OF
		cRFD_STA_Error: 
			getCmdState := 'cRFD_STA_Error';
		cRFD_STA_WaitForJob: 
			getCmdState := 'cRFD_STA_WaitForJob';
		cRFD_STA_PowerOnBusy: 
			getCmdState := 'cRFD_STA_PowerOnBusy';
		cRFD_STA_OffBusy: 
			getCmdState := 'cRFD_STA_OffBusy';
		cRFD_STA_Off: 
			getCmdState := 'cRFD_STA_Off';
		cRFD_STA_WriteBusy: 
			getCmdState := 'cRFD_STA_WriteBusy';
		cRFD_STA_ReadBusy: 
			getCmdState := 'cRFD_STA_ReadBusy';
		cRFD_STA_TagInitBusy: 
			getCmdState := 'cRFD_STA_TagInitBusy';
		cRFD_STA_CheckBusy: 
			getCmdState := 'cRFD_STA_CheckBusy';
		cRFD_STA_MDSBusy: 
			getCmdState := 'cRFD_STA_MDSBusy';
		cRFD_STA_SLGBusy: 
			getCmdState := 'cRFD_STA_SLGBusy';

	END_CASE;
END_IF
END_METHOD

METHOD getSIf : POINTER TO T_RFD
getSIf := ADR(SIf);
END_METHOD

METHOD PROTECTED sta_CheckBusy : BOOL
// state implemetation
//--------------------------------------------------------------------------------------
// Entry action
	IF (stStateMachine.intState<>stStateMachine.intStateLastCycle) THEN
		stStateMachine.intStateLastCycle := stStateMachine.intState;
			// Byte 0 => Lenght
			aTxData[0] := 2;
			// Byte 1 => Command read 4=single; 14=continious
			aTxData[1] := 16#FF;
			// Byte 2 => Spare
			aTxData[2] := 0;
						
			udiComSizeSendData := 3;
			bolComSend := TRUE;	
			SIf.stStatus.bolL_UEB := FALSE;
	END_IF


//--------------------------------------------------------------------------------------
// Cyclic action
	IF (stStateMachine.intState=stStateMachine.intStateLastCycle) THEN

		
		// State Change Condition
		IF (SIf.stErr.bolErrorActive = TRUE) THEN
			stStateMachine.intStateNext := cRFD_STA_Error;
		ELSIF (SIf.stStatus.bolL_UEB = TRUE) THEN
			stStateMachine.intStateNext := cRFD_STA_WaitForJob;
		END_IF
		
	END_IF

//--------------------------------------------------------------------------------------
// Exit action
	IF (stStateMachine.intState<>stStateMachine.intStateNext) THEN
		SIf.intCmd := cRFD_CMD_DONE;
	END_IF
END_METHOD

METHOD PROTECTED sta_Error : BOOL
// state implemetation
//--------------------------------------------------------------------------------------
// Entry action
	IF (stStateMachine.intState<>stStateMachine.intStateLastCycle) THEN
		stStateMachine.intStateHistory := stStateMachine.intStateLastCycle;
		stStateMachine.intStateLastCycle := stStateMachine.intState;
		
		SIf.stErr.bolErrorActive := TRUE;
		IF (SIf.stErr.bolComError = TRUE) OR (SIf.stErr.bolProtcolError = TRUE) THEN
			; //Written in different settings
		ELSIF SIf.stErr.bolSDOError = TRUE THEN
			SIf.stErr.udiErrorID := udiSdoErrorNbr;
		ELSIF SIf.stErr.bolRFIDError = TRUE THEN	
			SIf.stErr.udiErrorID := 1000 * aRxData[1] + bytRFIDState;
		ELSIF (udiResetCount >=SIf.stCfg.udiRetry) OR (udiJobCount >= SIf.stCfg.udiRetry) THEN
			SIf.stErr.udiErrorID := SIf.stCfg.udiRetry;
		ELSE
			SIf.stErr.udiErrorID := 0;
		END_IF


	END_IF


//--------------------------------------------------------------------------------------
// Cyclic action
	IF (stStateMachine.intState=stStateMachine.intStateLastCycle) THEN
		
		// State Change Condition
		IF (SIf.stErr.bolErrAck = TRUE) THEN
			// Reset all active errors
			SIf.stErr.bolErrorActive := FALSE;
			SIf.stErr.bolRFIDError := FALSE;
			SIf.stErr.bolComError := FALSE;
			SIf.stErr.bolProtcolError := FALSE;
			SIf.stErr.bolSDOError := FALSE;
			SIf.stErr.udiErrorID := 0;
			bolComSend := FALSE;
			SIf.stStatus.bolInitOk := FALSE;
			SIf.stStatus.bolOn := FALSE;
			SIf.stStatus.bolStartupOk := FALSE;
			SIf.stStatus.bolPresent := FALSE;
			SIf.stErr.bolErrAck := FALSE;
			
//			IF stStateMachine.intStateHistory < cRFD_STA_WaitForJob THEN
				stStateMachine.intStateNext := cRFD_STA_Off;
			//ELSE
			//	stStateMachine.intStateNext := cRFD_STA_WaitForJob;		
//			END_IF
		END_IF
	END_IF




//--------------------------------------------------------------------------------------
// Exit action
	IF (stStateMachine.intState<>stStateMachine.intStateNext) THEN
		;
	END_IF
END_METHOD

METHOD PROTECTED sta_MDSBusy : BOOL
// state implemetation
//--------------------------------------------------------------------------------------
// Entry action
	IF (stStateMachine.intState<>stStateMachine.intStateLastCycle) THEN
		stStateMachine.intStateLastCycle := stStateMachine.intState;
			stSubStateMachine.intState := cRFD_SUB_Write1;
			stSubStateMachine.intStateNext := cRFD_SUB_Write1;
	END_IF


//--------------------------------------------------------------------------------------
// Cyclic action
	IF (stStateMachine.intState=stStateMachine.intStateLastCycle) THEN
		CASE stSubStateMachine.intState OF
			cRFD_SUB_Write1:
				// Byte 0 => Lenght
				aTxData[0] := 5;
				// Byte 1 => Command read 4=single; 14=continious
				aTxData[1] := 16#B;
				// Byte 2 => Spare
				aTxData[2] := 0;
				// Byte 3 => Mode
				aTxData[3] := 3;
				// Byte 4 => Spare
				aTxData[4] := 0;
				// Byte 5 => Spare
				aTxData[5] := 0; 

						
				udiComSizeSendData := 6;
				bolComSend := TRUE;	
				stSubStateMachine.intState := cRFD_SUB_Wait1;
		
			cRFD_SUB_Wait1:
				IF bolMDSJobDone = TRUE THEN
					stSubStateMachine.intState := cRFD_SUB_SubStatesEnd;
					bolMDSJobDone := FALSE;
				END_IF
		cRFD_SUB_SubStatesEnd:
				;
				
		END_CASE
		
		// State Change Condition
		IF (SIf.stErr.bolComError = TRUE) OR ((SIf.stErr.bolRFIDError = TRUE) AND (udiJobCount > SIf.stCfg.udiRetry)) THEN
			stStateMachine.intStateNext := cRFD_STA_Error;
		ELSIF (SIf.stErr.bolRFIDError = TRUE) THEN
			udiJobCount := udiJobCount + 1;
			stStateMachine.intStateLastCycle := 0; // Startcycle again
		ELSIF (stSubStateMachine.intState = cRFD_SUB_SubStatesEnd) THEN
			udiJobCount := 0;
			stStateMachine.intStateNext := cRFD_STA_WaitForJob;
		END_IF
		
	END_IF

//--------------------------------------------------------------------------------------
// Exit action
	IF (stStateMachine.intState<>stStateMachine.intStateNext) THEN
		SIf.intCmd := cRFD_CMD_DONE;
	END_IF
END_METHOD

METHOD PROTECTED sta_Off : BOOL
// state implemetation
//--------------------------------------------------------------------------------------
// Entry action
	IF (stStateMachine.intState<>stStateMachine.intStateLastCycle) THEN
		stStateMachine.intStateLastCycle := stStateMachine.intState;
		
	END_IF


//--------------------------------------------------------------------------------------
// Cyclic action
	IF (stStateMachine.intState=stStateMachine.intStateLastCycle) THEN

		
		// State Change Condition
		IF (FALSE) THEN
			stStateMachine.intStateNext := cRFD_STA_Error;
		ELSIF (SIf.intCmd<>RFD_Cmd.cRFD_CMD_DONE) THEN
			stStateMachine.intStateNext := cRFD_STA_PowerOnBusy;
		END_IF
		
	END_IF

//--------------------------------------------------------------------------------------
// Exit action
	IF (stStateMachine.intState<>stStateMachine.intStateNext) THEN
		;
	END_IF
END_METHOD

METHOD PROTECTED sta_OffBusy : BOOL
// state implemetation
//--------------------------------------------------------------------------------------
// Entry action
	IF (stStateMachine.intState<>stStateMachine.intStateLastCycle) THEN
		stStateMachine.intStateLastCycle := stStateMachine.intState;
			IF SIf.stStatus.bolOn = TRUE THEN
				stSubStateMachine.intState := cRFD_SUB_Prepare;		// First Time set Baudrate and communication Settings
				stSubStateMachine.intStateNext := cRFD_SUB_Prepare;		// First Time set Baudrate and communication Settings
			ELSE
				stSubStateMachine.intState := cRFD_SUB_SubStatesEnd;
				stSubStateMachine.intStateNext := cRFD_SUB_SubStatesEnd;
			END_IF
			bolAntennaJobDone := FALSE;
	END_IF


//--------------------------------------------------------------------------------------
// Cyclic action
	IF (stStateMachine.intState=stStateMachine.intStateLastCycle) THEN
		
		// main statemachine of base controller
		CASE stSubStateMachine.intState OF
			cRFD_SUB_Prepare: 
				FOR udiI := 0 TO SIZEOF(aTxData) DO
					aTxData[udiI] := 0;
				END_FOR
				
				/// Send Command to set antenna OFF
				// Byte 0 => Lenght of telegram
				aTxData[0] := 3;
				// Byte 1 => Command Antenna job
				aTxData[1] := 16#A;
				// Byte 2 => Spare
				aTxData[2] := 0;
				// Byte 3 => Mode 1=On; 2=Off
				aTxData[3] := 2;
				
				udiComSizeSendData := 4;
				bolComSend := TRUE;
				stSubStateMachine.intStateNext := cRFD_SUB_SendBusy;
		
		cRFD_SUB_SendBusy:		
				IF ((SIf.stErr.bolComError = FALSE) AND (bolComSend = FALSE)) THEN
					stSubStateMachine.intStateNext := cRFD_SUB_WaitAnswer;
				END_IF

			cRFD_SUB_WaitAnswer:
				IF (bolAntennaJobDone = TRUE) THEN
					SIf.stStatus.bolOn := FALSE;
					stSubStateMachine.intStateNext := cRFD_SUB_SubStatesEnd;
				END_IF
				
			cRFD_SUB_SubStatesEnd:
				;
		END_CASE
		
		stSubStateMachine.intStateLastCycle := stSubStateMachine.intState;
		IF (stSubStateMachine.intState<>stSubStateMachine.intStateNext) THEN
			stSubStateMachine.intState := stSubStateMachine.intStateNext;  // set next state for next cycle
		END_IF
		

		// State Change Condition
		IF (stSubStateMachine.intStateNext = cRFD_SUB_SubStatesEnd) THEN
			stStateMachine.intStateNext := cRFD_STA_Off;
		END_IF
		
	END_IF


//--------------------------------------------------------------------------------------
// Exit action
	IF (stStateMachine.intState<>stStateMachine.intStateNext) THEN
		SIf.intCmd := cRFD_CMD_DONE;
		SIf.stStatus.bolOn := FALSE;
	END_IF
END_METHOD

METHOD PROTECTED sta_PowerOnBusy : BOOL
// state implemetation
//--------------------------------------------------------------------------------------
// Entry action
	IF (stStateMachine.intState<>stStateMachine.intStateLastCycle) THEN
		stStateMachine.intStateLastCycle := stStateMachine.intState;

			// original set parameter to RFID
			IF bolInitComDone=FALSE THEN
				//stSubStateMachine.intState := cRFD_SUB_SetBaudrate;		// First Time set Baudrate and communication Settings
				//stSubStateMachine.intStateNext := cRFD_SUB_SetBaudrate;		// First Time set Baudrate and communication Settings
				// pre 2013-10-11 Not setting Baudrate because this is done in HW Configuration
				stSubStateMachine.intState := cRFD_SUB_ClearBuffer;
				stSubStateMachine.intStateNext := cRFD_SUB_ClearBuffer;
			ELSE
				stSubStateMachine.intState := cRFD_SUB_ClearBuffer;
				stSubStateMachine.intStateNext := cRFD_SUB_ClearBuffer;
			END_IF

			bolSdoExecute := FALSE;
			bolResetJobDone := FALSE;
			fbTimeoutState.IN := FALSE;
			fbTimeoutState.PT := T#5S;
			fbTimeoutState();
			fbTimeoutState.IN := TRUE;
	END_IF


//--------------------------------------------------------------------------------------
// Cyclic action
	IF (stStateMachine.intState=stStateMachine.intStateLastCycle) THEN
		
		// main statemachine of base controller
		CASE stSubStateMachine.intState OF
			cRFD_SUB_SetBaudrate:
				IF stSubStateMachine.intStateLastCycle <> stSubStateMachine.intState THEN
					stSubStateMachine.intStateLastCycle := stSubStateMachine.intState;
				END_IF
				fbEcCoeSdoWrite(
					sNetId:= SIf.stCfg.stNetId, 
					nSlaveAddr:= SIf.stCfg.uinSlaveAddr, 
					nIndex:= SIf.stCfg.uinCoeIndexComSettings, 
					nSubIndex:= SIf.stCfg.usiCoeSubindexComBaudrate, 
					pSrcBuf:= ADR(SIf.stCfg.uinBaudrate), 
					cbBufLen:= SIZEOF(SIf.stCfg.uinBaudrate), 
					bExecute:= bolSdoExecute, 
					tTimeout:= DEFAULT_ADS_TIMEOUT, 
					bBusy=> bolSdoBusy, 
					bError=> SIf.stErr.bolSDOError, 
					nErrId=> udiSdoErrorNbr);
					
					
				IF 	(bolSdoExecute = TRUE) THEN
					IF ((SIf.stErr.bolSDOError = FALSE) AND (bolSdoBusy = FALSE)) THEN
						bolSdoExecute := FALSE;
						stSubStateMachine.intStateNext := cRFD_SUB_ClearBuffer;
					END_IF
				ELSE
					bolSdoExecute := TRUE;
				END_IF
				
			
			cRFD_SUB_SetComSettings:
				IF stSubStateMachine.intStateLastCycle <> stSubStateMachine.intState THEN
					stSubStateMachine.intStateLastCycle := stSubStateMachine.intState;
				END_IF
				fbEcCoeSdoWrite(
					sNetId:= SIf.stCfg.stNetId, 
					nSlaveAddr:= SIf.stCfg.uinSlaveAddr, 
					nSubIndex:= SIf.stCfg.usiCoeSubindexComDataframe, 
					nIndex:= SIf.stCfg.uinCoeIndexComSettings, 
					pSrcBuf:= ADR(SIf.stCfg.uinComSettings), 
					cbBufLen:= SIZEOF(SIf.stCfg.uinComSettings), 
					bExecute:= bolSdoExecute, 
					tTimeout:= T#2S, 
					bBusy=> bolSdoBusy, 
					bError=> SIf.stErr.bolSDOError, 
					nErrId=> udiSdoErrorNbr);
					
				IF 	(bolSdoExecute = TRUE) THEN
					IF ((SIf.stErr.bolSDOError = FALSE) AND (bolSdoBusy = FALSE)) THEN
						bolSdoExecute := FALSE;
						stSubStateMachine.intStateNext := cRFD_SUB_ClearBuffer;
					END_IF
				ELSE
					bolSdoExecute := TRUE;
				END_IF

	
			cRFD_SUB_ClearBuffer: 	 
				IF stSubStateMachine.intStateLastCycle <> stSubStateMachine.intState THEN
					stSubStateMachine.intStateLastCycle := stSubStateMachine.intState;
				END_IF
				bolInitComDone := TRUE;
				IF (SIf.stErr.bolComError = FALSE) THEN
					stSubStateMachine.intStateNext := cRFD_SUB_InitString;
				END_IF

				
			cRFD_SUB_InitString: 
				IF stSubStateMachine.intStateLastCycle <> stSubStateMachine.intState THEN
					stSubStateMachine.intStateLastCycle := stSubStateMachine.intState;
					aTxData[0] := 10;
					// Byte 1 => Spare
					aTxData[1] := 0;
					// Byte 2 => Spare
					aTxData[2] := 0;
					// Byte 3 => Spare
					aTxData[3] := 0;
					// Byte 4 => Reset Parameter
					aTxData[4] := 16#25; // SIf.stCfg.usiResetParameter;
					// Byte 5 => Reset option
					aTxData[5] := 16#2; //SIf.stCfg.usiResetOption1;
					// Byte 6 => dili = Setting of sendepower antenna (only RF380R)
					aTxData[6] := 0; //0;
					// Byte 7 => Spare
					aTxData[7] := 0;
					// Byte 8 => mtag = Maximal value of tags in field
					aTxData[8] := 1;
					// Byte 9 => Spare
					aTxData[9] := 0;
					// Byte 10 => ftim = Setting for the Air interface
					aTxData[10] := 1;
					
					udiComSizeSendData := 11;
					bolComSend := TRUE;
				END_IF
			
				IF ((SIf.stErr.bolComError = 0) AND (bolComSend = FALSE)) THEN	 //AND (bolComSendBusy_old = TRUE)
					stSubStateMachine.intStateNext := cRFD_SUB_CheckPon;
				END_IF

			cRFD_SUB_CheckPon:
				IF (bolResetJobDone = TRUE) THEN
					stSubStateMachine.intStateNext := cRFD_SUB_SubStatesEnd;
				ELSIF (bolResetJobError =TRUE) AND (udiResetCount < SIf.stCfg.udiRetry) THEN
					bolResetJobError := FALSE;
					udiResetCount := udiResetCount + 1;
					stSubStateMachine.intStateNext := cRFD_SUB_InitString;
				END_IF
				
			cRFD_SUB_SubStatesEnd:
				;
		END_CASE
		
		stSubStateMachine.intStateLastCycle := stSubStateMachine.intState;
		fbTimeoutState();
		// Check Timeout of communication
		IF fbTimeoutState.Q = TRUE THEN
			SIf.stErr.bolComError := TRUE;
			SIf.stErr.udiErrorID := TIME_TO_UDINT(fbTimeoutState.ET);
		END_IF
		
		IF udiResetCount >= SIf.stCfg.udiRetry THEN
			SIf.stErr.bolComError := TRUE;
			SIf.stErr.udiErrorID := udiResetCount;
		END_IF

		IF (stSubStateMachine.intState<>stSubStateMachine.intStateNext) THEN
			stSubStateMachine.intState := stSubStateMachine.intStateNext;  // set next state for next cycle
			//stSubStateMachine.udiTimeInState_ms := 0; // reset timer
			// log state change -> open point
		//ELSE
			// increment time in state	
			//stSubStateMachine.intStateLastCycle := stSubStateMachine.udiTimeInState_ms + me.FUBInfo.udiSample_ms;
		END_IF
		

		// State Change Condition
		IF (SIf.stErr.bolComError = TRUE) OR (SIf.stErr.bolSDOError = TRUE) THEN
			stStateMachine.intStateNext := cRFD_STA_Error;
		ELSIF (stSubStateMachine.intStateNext = cRFD_SUB_SubStatesEnd) THEN
			stStateMachine.intStateNext := cRFD_STA_WaitForJob;
		END_IF
		
	END_IF


//--------------------------------------------------------------------------------------
// Exit action
	IF (stStateMachine.intState<>stStateMachine.intStateNext) THEN
		SIf.intCmd := cRFD_CMD_DONE;
		SIf.stStatus.bolStartupOk := TRUE;
		SIf.stStatus.bolInitOk := TRUE;
		SIf.stStatus.bolOn := TRUE;
	END_IF
END_METHOD

METHOD PROTECTED sta_ReadBusy : BOOL
// state implemetation
//--------------------------------------------------------------------------------------
// Entry action
	IF (stStateMachine.intState<>stStateMachine.intStateLastCycle) THEN
		stStateMachine.intStateLastCycle := stStateMachine.intState;
			// Byte 0 => Lenght
			aTxData[0] := 5;
			// Byte 1 => Command read 2=single; 12=continious
			aTxData[1] := 2;
			// Byte 2 => Spare
			aTxData[2] := 0;
			// Byte 3 => Adress MSB
			uinValue := SIf.stCur.uinAdressTag;
			uinValue := ROL(uinValue,8);
			aTxData[3] := UINT_TO_USINT(uinValue);
			// Byte 4 => Adress LSB
			aTxData[4] := UINT_TO_USINT(SIf.stCur.uinAdressTag);
			// Byte 5 =>Lenght
			aTxData[5] := SIf.stCur.usiCount; 
					
			udiComSizeSendData := 6;
			bolComSend := TRUE;	
	END_IF


//--------------------------------------------------------------------------------------
// Cyclic action
	IF (stStateMachine.intState=stStateMachine.intStateLastCycle) THEN


		
		// State Change Condition
		IF (SIf.stErr.bolComError = TRUE) OR ((SIf.stErr.bolRFIDError = TRUE) AND (udiJobCount > SIf.stCfg.udiRetry)) THEN
			stStateMachine.intStateNext := cRFD_STA_Error;
		ELSIF (SIf.stErr.bolRFIDError = TRUE) THEN
			udiJobCount := udiJobCount + 1;
			stStateMachine.intStateLastCycle := 0; // Startcycle again
		ELSIF ((SIf.stErr.bolComError = 0) AND (bolReadDone = TRUE)) THEN
			bolReadDone := FALSE;
			udiJobCount := 0;
			stStateMachine.intStateNext := cRFD_STA_WaitForJob;
		END_IF
		
	END_IF

//--------------------------------------------------------------------------------------
// Exit action
	IF (stStateMachine.intState<>stStateMachine.intStateNext) THEN
		SIf.intCmd := cRFD_CMD_DONE;
	END_IF
END_METHOD

METHOD PROTECTED sta_SLGBusy : BOOL
// state implemetation
//--------------------------------------------------------------------------------------
// Entry action
	IF (stStateMachine.intState<>stStateMachine.intStateLastCycle) THEN
		stStateMachine.intStateLastCycle := stStateMachine.intState;
			stSubStateMachine.intState := cRFD_SUB_Write1;
			stSubStateMachine.intStateNext := cRFD_SUB_Write1;
	END_IF


//--------------------------------------------------------------------------------------
// Cyclic action
	IF (stStateMachine.intState=stStateMachine.intStateLastCycle) THEN
		CASE stSubStateMachine.intState OF
			cRFD_SUB_Write1:
				// Byte 0 => Lenght
				aTxData[0] := 6;
				// Byte 1 => Command read 4=single; 14=continious
				aTxData[1] := 4;
				// Byte 2 => Spare
				aTxData[2] := 0;
				// Byte 3 => Mode
				aTxData[3] := 1;
				// Byte 4 => Spare
				aTxData[4] := 0;
				// Byte 5 => Spare
				aTxData[5] := 0; 
				// Byte 6 => Spare
				aTxData[6] := 0; 
						
				udiComSizeSendData := 7;
				bolComSend := TRUE;	
				stSubStateMachine.intState := cRFD_SUB_Wait1;
		
			cRFD_SUB_Wait1:
				IF bolSLGJobDone = TRUE THEN
					stSubStateMachine.intState := cRFD_SUB_Write6;
					bolSLGJobDone := FALSE;
				END_IF
			cRFD_SUB_Write6:
				// Byte 0 => Lenght
				aTxData[0] := 6;
				// Byte 1 => Command read 4=single; 14=continious
				aTxData[1] := 4;
				// Byte 2 => Spare
				aTxData[2] := 0;
				// Byte 3 => Mode
				aTxData[3] := 6;
				// Byte 4 => Spare
				aTxData[4] := 0;
				// Byte 5 => Spare
				aTxData[5] := 0; 
				// Byte 6 => Spare
				aTxData[6] := 0; 
						
				udiComSizeSendData := 7;
				bolComSend := TRUE;	
				stSubStateMachine.intState := cRFD_SUB_Wait6;
		
			cRFD_SUB_Wait6:
				IF bolSLGJobDone = TRUE THEN
					stSubStateMachine.intState := cRFD_SUB_SubStatesEnd;
					bolSLGJobDone := FALSE;
				END_IF
			
			cRFD_SUB_SubStatesEnd:
				;
				
		END_CASE
		
		// State Change Condition
		IF (SIf.stErr.bolComError = TRUE) OR ((SIf.stErr.bolRFIDError = TRUE) AND (udiJobCount > SIf.stCfg.udiRetry)) THEN
			stStateMachine.intStateNext := cRFD_STA_Error;
		ELSIF (SIf.stErr.bolRFIDError = TRUE) THEN
			udiJobCount := udiJobCount + 1;
			stStateMachine.intStateLastCycle := 0; // Startcycle again
		ELSIF (stSubStateMachine.intState = cRFD_SUB_SubStatesEnd) THEN
			udiJobCount := 0;
			stStateMachine.intStateNext := cRFD_STA_WaitForJob;
		END_IF
		
	END_IF

//--------------------------------------------------------------------------------------
// Exit action
	IF (stStateMachine.intState<>stStateMachine.intStateNext) THEN
		SIf.intCmd := cRFD_CMD_DONE;
	END_IF
END_METHOD

METHOD PROTECTED sta_TagInitBusy : BOOL
// state implemetation
//--------------------------------------------------------------------------------------
// Entry action
	IF (stStateMachine.intState<>stStateMachine.intStateLastCycle) THEN
		stStateMachine.intStateLastCycle := stStateMachine.intState;
		
	END_IF


//--------------------------------------------------------------------------------------
// Cyclic action
	IF (stStateMachine.intState=stStateMachine.intStateLastCycle) THEN

		
		// State Change Condition
		IF (FALSE) THEN
			stStateMachine.intStateNext := cRFD_STA_Error;
		ELSIF (TRUE) THEN
			stStateMachine.intStateNext := cRFD_STA_WaitForJob;
		END_IF
		
	END_IF

//--------------------------------------------------------------------------------------
// Exit action
	IF (stStateMachine.intState<>stStateMachine.intStateNext) THEN
		IF SIf.intCmd = stStateMachine.intState THEN
			SIf.intCmd := cRFD_CMD_DONE;
		END_IF
	END_IF
END_METHOD

METHOD PROTECTED sta_WaitForJob : BOOL
// state implemetation
//--------------------------------------------------------------------------------------
// Entry action
	IF (stStateMachine.intState<>stStateMachine.intStateLastCycle) THEN
		stStateMachine.intStateLastCycle := stStateMachine.intState;
		
	END_IF


